			tTimeToDose := REAL_TO_TIME( (UINT_TO_REAL(nDoseQtyMls) * 1000.0) / (UINT_TO_REAL(nDoseRateMLph) / 60.0 / 60.0 ));
			fbTONdoseTime.IN := FALSE;
			fbTONdoseTime.PT := tTimeToDose;
			fbTONdoseTime.IN := TRUE;
			eState := E_DeviceState.RUNNING;
			bBusy := TRUE;
			eSMState := WAIT;
		END_IF
		
		IF fbTONdoseTime.Q THEN
			eStateTarget := E_DeviceState.IDLE;
			eState := E_DeviceState.IDLE;
			bBusy := FALSE;
		END_IF
			
	END_IF

{warning 'add method implementation '}
METHOD disable : BOOL
bEnable := False;
END_METHOD

{warning 'add method implementation '}
METHOD enable : BOOL
bEnable := True;
END_METHOD

{warning 'add method implementation '}
METHOD executeDose : BOOL
VAR_INPUT
	DoseQtyMls	: UINT;
	DoseRateMlph	: UINT;
	RequestComplete	: POINTER TO BOOL;
END_VAR
VAR_OUTPUT
	RequestAccepted	: BOOL;
END_VAR
IF bBusy = FALSE THEN
	IF bEnable THEN
		nDoseQtyMls := DoseQtyMls;
		nDoseRateMLph := DoseRateMLph;
		tTimeToDose := REAL_TO_TIME( (UINT_TO_REAL(nDoseQtyMls) * 1000.0) / (UINT_TO_REAL(DoseRateMLph) / 60.0 / 60.0 ));
		RequestAccepted := TRUE;
		bRequestSentToMaster := FALSE;
		bRequestFinished := RequestComplete;
		eSMState := SET_DOSE_TRIG;
		executeDose := TRUE;
	END_IF
ELSE
	executeDose := FALSE;
END_IF
END_METHOD

METHOD FB_init : BOOL
VAR_INPUT
	bInitRetains : BOOL; // if TRUE, the retain variables are initialized (warm start / cold start)
	bInCopyCode : BOOL;  // if TRUE, the instance afterwards gets moved into the copy code (online change)
	
	MotorID: STRING;
	MotorDescr: STRING;
	
	ModbusUnitID: UINT; 
	//ModbusMaster: FB_ModbusMaster;
	
END_VAR
sID := MotorID;
sDescr := MotorDescr;
nModbusUnitID := ModbusUnitID;
//fbModbusMaster := ModbusMaster;
END_METHOD

METHOD readReg : BOOL
VAR_INPUT
	RequestComplete	: POINTER TO BOOL;
	AddressToRead: UINT;
	NumberWords: UINT;
END_VAR
VAR_OUTPUT
	RequestAccepted	: BOOL;
END_VAR
IF bBusy = FALSE THEN
	IF bEnable THEN
		nReadRegsVals[1] := 16#00;
		nReadRegsVals[2] := 16#00;
		nReadRegsVals[3] := 16#00;
		nReadRegsVals[4] := 16#00;
		nRegisterWordstoRead := NumberWords;
		nAddrRead:= AddressToRead;
		eSMState := READ_TRIG;
		bBusy := TRUE;		
		readReg := TRUE;		
	END_IF
ELSE
	readReg := FALSE;
END_IF
END_METHOD

METHOD resetStatistics : BOOL
VAR_INPUT
END_VAR
END_METHOD

{warning 'add method implementation '}
METHOD setBatch : BOOL
VAR_INPUT
	BatchQtyMl	: UINT;
	RequestComplete	: POINTER TO BOOL;
END_VAR
VAR_OUTPUT
	RequestAccepted	: BOOL;
END_VAR

VAR
	SET_BATCH_QTY_TRIG: E_DeviceState;
END_VAR
IF bBusy = FALSE THEN
	IF bEnable THEN
		nBatchQtyMl := BatchQtyMl;
		RequestAccepted := TRUE;
		bRequestSentToMaster := FALSE;
		bRequestFinished := RequestComplete;
		eSMState := SET_BATCH_QTY_TRIG;
		setBatch := TRUE;
	END_IF
ELSE 
	setBatch := FALSE;
END_IF
END_METHOD

METHOD setCapacity : BOOL
VAR_INPUT
	Capacity: DINT;
END_VAR
VAR_INPUT
	RequestComplete	: POINTER TO BOOL;
END_VAR
VAR_OUTPUT
	RequestAccepted	: BOOL;
END_VAR
IF bBusy = FALSE THEN
	IF bEnable THEN
		nWriteRegsVals[1] := DINT_TO_WORD(Capacity);
		nQtyWordsWrite := 1;
		nAddrWrite := 16#C1;
		eSMState := WRITE_TRIG;
		bBusy := TRUE;		
		setCapacity := TRUE;		
	END_IF
ELSE
	setCapacity := FALSE;
END_IF
END_METHOD

METHOD setDoseParams : BOOL
VAR_INPUT
	DoseQtyMls	: UINT;
	DoseRateMlph	: UINT;
END_VAR

nDoseQtyMls := DoseQtyMls;
nDoseRateMLph := DoseRateMlph;
END_METHOD

METHOD setModbusMaster : BOOL
VAR_INPUT
	ModbusMaster: FB_ModbusMaster;
END_VAR

fbModbusMaster REF= ModbusMaster;
END_METHOD

{warning 'add method implementation '}
METHOD setOFF : BOOL
VAR_INPUT
	RequestComplete	: POINTER TO BOOL;
END_VAR
VAR_OUTPUT
	RequestAccepted	: BOOL;
END_VAR
IF bBusy = FALSE THEN
	IF bEnable THEN
		nWriteRegsVals[1] := 16#0;
		nQtyWordsWrite := 1;
		nAddrWrite := 16#8C;
		eSMState := WRITE_TRIG;
		bBusy := TRUE;		
		setOFF := TRUE;		
	END_IF
ELSE
	setOFF := FALSE;
END_IF
END_METHOD

{warning 'add method implementation '}
METHOD setON : BOOL
VAR_INPUT
	RateMlph	: UINT;
	RequestComplete	: POINTER TO BOOL;
END_VAR
VAR_OUTPUT
	RequestAccepted	: BOOL;
END_VAR
IF bBusy = FALSE AND bEnable THEN
	nWriteRegsVals[1] := 16#1;
	nQtyWordsWrite := 1;
	nAddrWrite := 16#8C;		// Emec have 2 different Modbus register schemes (check which version the pumps are and amend if necessary)
	eSMState := WRITE_TRIG;
	bBusy := TRUE;
	setON := TRUE;
ELSE
	setON := FALSE;
END_IF
END_METHOD

METHOD writeReg : BOOL
VAR_INPUT
	RequestComplete	: POINTER TO BOOL;
	Register: WORD;
	Value: WORD;
END_VAR
VAR_OUTPUT
	RequestAccepted	: BOOL;
END_VAR
IF bBusy = FALSE THEN
	IF bEnable THEN
		nWriteRegsVals[1] := Value;
		nQtyWordsWrite := 1;
		nAddrWrite := Register;
		eSMState := WRITE_TRIG;
		bBusy := TRUE;				
	END_IF
END_IF
END_METHOD

END_FUNCTION_BLOCK

// ---- POUs/99 Utilities/_ss/FB_ModbusMaster.TcPOU
FUNCTION_BLOCK FB_ModbusMaster

VAR
	MB: ModbusRtuMaster_KL6x22B;
	
	nReadRegsVals: POINTER TO ARRAY[1..10] OF WORD;
	nWriteRegVals: ARRAY[1..10] OF WORD;
	
	
	bRequestFinshed : POINTER TO BOOL;
		
	nSlaveAddress : BYTE;
	nQtyWordsToRead : WORD;
	nQtyWordsToWrite : WORD;
	nAdrFirstSlaveRegisterRead : WORD;
	nAdrFirstSlaveRegisterWrite : WORD;
	nTimeout : TIME := T#5S;
	
	
	// State Machine
	eState: (IDLE, BUSY, ERROR) := IDLE;
	eSMtate: (WAIT, READ_TRIG, READ, WRITE_TRIG, WRITE, ERROR) := WAIT;
	eSMState_prev:  (WAIT, READ_TRIG, READ, WRITE_TRIG, WRITE, ERROR) := WAIT;
	bBusy: BOOL;
	
	//eOperationType: (READ_OP, WRITE_OP, READWRITE_OP);
	eOperationType: E_AccessType;
	fbTrigger : R_TRIG;
	
	bOperationFirstRun: BOOL := TRUE;
	nNumRetries: INT := 0; 
	nRetryThreshold: INT := 10;

END_VAR

fbTrigger();

CASE eState OF
	WAIT :
		eState := IDLE;
		MB.ReadRegs(Execute := FALSE);
        MB.WriteRegs(Execute := FALSE);
	
		
		IF fbTrigger.Q THEN
			IF eOperationType = E_AccessType.WRITE THEN
				eSMtate := WRITE_TRIG;
			ELSIF eOperationType = E_AccessType.READ THEN
				eSMtate := READ_TRIG;
			END_IF
		END_IF
		
		
		
	READ_TRIG : 
		eState := BUSY;
		IF bOperationFirstRun THEN
			nNumRetries := 0;
			bOperationFirstRun := FALSE;
		END_IF
	
		IF eOperationType = E_AccessType.READ THEN
			
			 MB.ReadRegs(
				UnitID:= nSlaveAddress, 
				Quantity:= nQtyWordsToRead, 
				MBAddr:= nAdrFirstSlaveRegisterRead, 
				cbLength:= nQtyWordsToRead * 2,//SIZEOF(nReadRegsVals), 
				pMemoryAddr:= ADR(nReadRegsVals), 
				Execute:= TRUE, 
				Timeout:= nTimeout );
			
			
			IF NOT MB.BUSY THEN 
				MB.ReadRegs(Execute := FALSE );
				bBusy := TRUE;
				IF MB.Error THEN 
					eSMState_prev := eSMtate;
					eSMtate := ERROR;           // handle errors 
				ELSE 
					eSMtate := READ; // [...]               // keep going 
				END_IF
			END_IF
		END_IF
		
		
	READ :
	
		IF NOT MB.BUSY THEN
			eSMtate := WAIT;
			bRequestFinshed^ := TRUE;
			bBusy := FALSE;
			fbTrigger.CLK := FALSE;
			bOperationFirstRun := TRUE;
		ELSIF MB.Error THEN
			eSMState_prev := eSMtate;
			eSMtate := ERROR;
		END_IF
	
	
	
	WRITE_TRIG :

		IF bOperationFirstRun THEN
			nNumRetries := 0;
			bOperationFirstRun := FALSE;
		END_IF
	(*
		MB.WriteRegs(
			UnitID:= nSlaveAddress, 
			Quantity:= nQtyWordsToWrite, 
			MBAddr:= nAdrFirstSlaveRegisterWrite, 
			cbLength:= nQtyWordsToWrite * 2, 
			pMemoryAddr:= ADR(nWriteRegVals), 
			Execute:= TRUE, 
			Timeout:= nTimeout); 
		*)	
		
		MB.UnitID:= nSlaveAddress;
		MB.Quantity:=1;
		MB.MBAddr:= nAdrFirstSlaveRegisterWrite;
		MB.cbLength:= nQtyWordsToWrite * 2;
		MB.pMemoryAddr:= ADR(nWriteRegVals);
		MB.Execute:= TRUE;
		MB.Timeout:= nTimeout;
		MB.WriteSingleRegister();
		
			
		IF NOT MB.BUSY THEN 
			//MB.WriteRegs(Execute := FALSE );
			MB.Execute := FALSE;
			bBusy := TRUE;
			IF MB.Error THEN 
				eSMState_prev := eSMtate;
				eSMtate := ERROR;           				// handle errors 
			ELSE 
				eSMtate := WRITE;			            // keep going 
			END_IF
		END_IF

	
		
	WRITE:
		IF NOT MB.BUSY THEN
			eSMtate := WAIT;
			bRequestFinshed^ := TRUE;
			bBusy := FALSE;
			fbTrigger.CLK := FALSE;
			bOperationFirstRun := TRUE;
		ELSIF MB.Error THEN
			eSMState_prev := eSMtate;
			eSMtate := ERROR;
		END_IF
	
		
	ERROR:
		nNumRetries := nNumRetries + 1;
		IF nNumRetries > nRetryThreshold THEN
			eState := ERROR;
		ELSE
			eSMtate := eSMState_prev;
		END_IF
		 
			
		

END_CASE

METHOD Error : BOOL
VAR_INPUT
END_VAR
Error := MB.Error;
END_METHOD

METHOD FB_init : BOOL
VAR_INPUT
	bInitRetains : BOOL; // if TRUE, the retain variables are initialized (warm start / cold start)
	bInCopyCode : BOOL;  // if TRUE, the instance afterwards gets moved into the copy code (online change)
END_VAR
END_METHOD

METHOD isBusy : BOOL
isBusy := bBusy;
END_METHOD

METHOD readRegs : BOOL
VAR_INPUT
	
	ReadRegsVals: POINTER TO ARRAY[1..10] OF WORD;
	SlaveAddress : UINT;
	QtyWordsToRead : UINT;
	AdrFirstSlaveRegisterRead : UINT;
	bRequestCompleted : POINTER TO BOOL;
	
END_VAR

VAR_OUTPUT
	bRequestAccepted: BOOL;
END_VAR
IF eState = WAIT THEN
	eOperationType := E_AccessType.READ;
	nReadRegsVals := ReadRegsVals;
	nSlaveAddress := UINT_TO_BYTE(SlaveAddress);
	nQtyWordsToRead := UINT_TO_WORD(QtyWordsToRead);
	nAdrFirstSlaveRegisterRead := UINT_TO_WORD(AdrFirstSlaveRegisterRead);
	fbTrigger.CLK := TRUE;
	bRequestAccepted := TRUE;
	bBusy := TRUE;
	bRequestFinshed := bRequestCompleted;
END_IF
END_METHOD

METHOD writeReg : BOOL
VAR_INPUT
	WriteRegVal: WORD;
	SlaveAddress : UINT;
	AdrFirstSlaveRegisterWrite : UINT;
	bRequestCompleted : POINTER TO BOOL;
END_VAR

VAR_OUTPUT
	bRequestAccepted: BOOL := FALSE;
END_VAR

IF eState = WAIT THEN
	eOperationType := E_AccessType.WRITE;
	nWriteRegVals[1] := WriteRegVal;
	nSlaveAddress := UINT_TO_BYTE(SlaveAddress);
	nQtyWordsToWrite := 1;
	nAdrFirstSlaveRegisterWrite := UINT_TO_BYTE(AdrFirstSlaveRegisterWrite);
	bRequestAccepted := TRUE;
	bRequestFinshed := bRequestCompleted;
	fbTrigger.CLK := TRUE;
	eState := WRITE_TRIG;
	
END_IF
END_METHOD

METHOD writeRegs : BOOL
VAR_INPUT

	WriteRegVals: ARRAY[1..10] OF WORD;
	
	SlaveAddress : UINT;
	QtyWordsToWrite : UINT;
	AdrFirstSlaveRegisterWrite : UINT;
	bRequestCompleted: POINTER TO BOOL;

END_VAR

VAR_OUTPUT
	bRequestAccepted: BOOL := FALSE;
END_VAR
IF eState = WAIT THEN
	eOperationType := E_AccessType.WRITE;
	nWriteRegVals := WriteRegVals;
	nSlaveAddress := UINT_TO_BYTE(SlaveAddress);
	nQtyWordsToWrite := UINT_TO_WORD(QtyWordsToWrite);
	nAdrFirstSlaveRegisterWrite := UINT_TO_WORD(AdrFirstSlaveRegisterWrite);
	fbTrigger.CLK := TRUE;
	bRequestAccepted := TRUE;
	bRequestFinshed := bRequestCompleted;
	eState := WRITE_TRIG;
END_IF
END_METHOD

END_FUNCTION_BLOCK

// ---- POUs/01 Actuators/Dosing Machine/FB_DrumFilter_Faivre120.TcPOU
{attribute 'OPC.UA.DA.StructuredType' := '1'}
FUNCTION_BLOCK FB_DrumFilter_Faivre120 EXTENDS FB_BaseDevice IMPLEMENTS I_Device

VAR
	
	{attribute 'OPC.UA.DA' := '1'}   
	bInContactor AT %I*: BOOL := FALSE;
	{attribute 'OPC.UA.DA' := '1'}   
	bOutContactor AT %Q*: BOOL := FALSE;
	{attribute 'OPC.UA.DA' := '1'}   
	bInMCCB AT %I*: BOOL := FALSE;
	{attribute 'OPC.UA.DA' := '1'}   
	bInRunning AT %I*: BOOL := FALSE;
	{attribute 'OPC.UA.DA' := '1'}   
	bInFault_Motors AT %I*: BOOL := FALSE;
	{attribute 'OPC.UA.DA' := '1'}   
	bInFault_Overflow AT %I*: BOOL := FALSE;
	{attribute 'OPC.UA.DA' := '0'}   
	eSMState: (WAIT, TURNING_ON, ON, TURNING_OFF, OFF);
	{attribute 'OPC.UA.DA' := '0'}   
	tActionTimeout: TIME := T#5S;
	{attribute 'OPC.UA.DA' := '0'}   
	fbTON_timeout: TON := (PT := tActionTimeout, IN := FALSE);
	{attribute 'OPC.UA.DA' := '0'}  
	fbTON_simulation_delay: TON := (PT := T#1S, IN := FALSE);
END_VAR

fbTONstartTime();
fbTONstopTime();


IF GVL.bAutoUpdateDeviceState THEN
	eState := eStateTarget;	
END_IF


IF eMode <> E_DeviceMode.SIMULATION THEN
	
	
	IF bEnable THEN
		IF eStateTarget = E_DeviceState.ON AND eState <> E_DeviceState.ON THEN
			eSMState := TURNING_ON;
		END_IF
	END_IF
	
	IF eStateTarget = E_DeviceState.OFF AND eState <> E_DeviceState.OFF THEN
			eSMState := TURNING_OFF;
	END_IF
	
	
	CASE eSMState OF
		
		WAIT:
			//Wait for method call to change ESMState
			
		TURNING_ON: 
			eState := E_DeviceState.TURNING_ON;
	
			bOutContactor := TRUE;
		
			IF fbTONstartTime.Q THEN
				eSMState := WAIT;
				raiseAlarm(Priority := E_AlarmPriority.High, Label := 'Failed to Start', Enabled := TRUE, DeviceAlarmID := 1);
			END_IF
			
			IF bInContactor  THEN
				eSMState := ON;
				eState := E_DeviceState.ON;
			END_IF
			
		ON:
			IF bInContactor <> TRUE THEN
				raiseAlarm(Priority := E_AlarmPriority.High, Label := 'Power Lost', Enabled := TRUE, DeviceAlarmID := 2);
				eState := E_DeviceState.OFF;
				eSMState := WAIT;
			END_IF
			
	
			
		TURNING_OFF:
			eState := E_DeviceState.TURNING_OFF;
			bOutContactor := FALSE;
	
					
			IF fbTONstopTime.Q THEN
				eSMState := WAIT;
				raiseAlarm(Priority := E_AlarmPriority.High, Label := 'Failed to Stop', Enabled := TRUE,  DeviceAlarmID := 3);
			END_IF 
			
			IF bInContactor = FALSE THEN
				eSMState := OFF;	
			END_IF
	
			
			
		OFF:
			eState := E_DeviceState.OFF;
			eSMState := WAIT;
			
			
	END_CASE
	
	
(*
				SIMULATION CODE 
				This code forces the contactor feedback ON or OFF depending on whether the device has been told to turn on or off
*)

ELSIF eMode = E_DeviceMode.SIMULATION THEN
	
fbTON_simulation_delay();
	
	IF eSMState = TURNING_ON THEN  					
		fbTON_simulation_delay.IN := TRUE;
		IF fbTON_simulation_delay.Q THEN
			bInContactor := TRUE;
			fbTON_simulation_delay.IN := FALSE;	
		END_IF
		
	ELSIF eSMState = TURNING_OFF THEN
		fbTON_simulation_delay.IN := TRUE;
		IF fbTON_simulation_delay.Q THEN
			bInContactor := FALSE;
			fbTON_simulation_delay.IN := FALSE;	
		END_IF
	END_IF
END_IF

{warning 'add method implementation '}
METHOD disable : BOOL
bEnable := FALSE;
END_METHOD

{warning 'add method implementation '}
METHOD enable : BOOL
bEnable := TRUE;
END_METHOD

METHOD FB_init : BOOL
VAR_INPUT
	bInitRetains : BOOL; // if TRUE, the retain variables are initialized (warm start / cold start)
	bInCopyCode : BOOL;  // if TRUE, the instance afterwards gets moved into the copy code (online change)
	
	FilterID: STRING(80);
	FIlterDescr: STRING(255);
END_VAR
sID := FilterID;
sDescr := FIlterDescr;
END_METHOD

METHOD setOff : BOOL
VAR_INPUT
END_VAR
eSMState := TURNING_OFF;
fbTONstopTime.IN := TRUE;
bBusy := FALSE;
END_METHOD

METHOD setOn : BOOL
VAR_INPUT
END_VAR
eSMState := TURNING_ON;
fbTONstartTime.IN := TRUE;
bBusy := TRUE;
END_METHOD

END_FUNCTION_BLOCK

// ---- POUs/01 Actuators/Dosing Machine/FB_DrumFilter_Faivre60.TcPOU
{attribute 'OPC.UA.DA.StructuredType' := '1'}
FUNCTION_BLOCK FB_DrumFilter_Faivre60 EXTENDS FB_BaseDevice IMPLEMENTS I_Device

VAR

	{attribute 'OPC.UA.DA' := '1'}   
	bInContactor AT %I*: BOOL := FALSE;
	{attribute 'OPC.UA.DA' := '1'}   
	bOutContactor AT %Q*: BOOL := FALSE;
	{attribute 'OPC.UA.DA' := '1'}   
	bInMCCB AT %I*: BOOL := FALSE;
	{attribute 'OPC.UA.DA' := '1'}   
	bInRunning AT %I*: BOOL := FALSE;
	{attribute 'OPC.UA.DA' := '1'}   
	bInFault_Motors AT %I*: BOOL := FALSE;
	{attribute 'OPC.UA.DA' := '1'}   
	bInFault_Overflow AT %I*: BOOL := FALSE;
	{attribute 'OPC.UA.DA' := '0'}   
	eSMState: (WAIT, TURNING_ON, ON, TURNING_OFF, OFF);
	{attribute 'OPC.UA.DA' := '0'}   
	tActionTimeout: TIME := T#5S;
	{attribute 'OPC.UA.DA' := '0'}   
	fbTON_timeout: TON := (PT := tActionTimeout, IN := FALSE);
	{attribute 'OPC.UA.DA' := '0'}
	fbTON_simulation_delay: TON := (PT := T#1S, IN := FALSE);
END_VAR

fbTONstartTime();
fbTONstopTime();

IF GVL.bAutoUpdateDeviceState THEN
	eState := eStateTarget;	
END_IF

IF eMode <> E_DeviceMode.SIMULATION THEN
	
	
	
	
	IF bEnable THEN
		IF eStateTarget = E_DeviceState.ON AND eState <> E_DeviceState.ON THEN
			eSMState := TURNING_ON;
		END_IF
	END_IF
	
	IF eStateTarget = E_DeviceState.OFF AND eState <> E_DeviceState.OFF THEN
			eSMState := TURNING_OFF;
	END_IF
	
	
	CASE eSMState OF
		
		WAIT:
			//Wait for method call to change ESMState
			
		TURNING_ON: 
			eState := E_DeviceState.TURNING_ON;
	
			bOutContactor := TRUE;
		
			IF fbTONstartTime.Q THEN
				eSMState := WAIT;
				raiseAlarm(Priority := E_AlarmPriority.High, Label := 'Failed to Start', Enabled := TRUE, DeviceAlarmID := 1);
			END_IF
			
			IF bInContactor  THEN
				eSMState := ON;
				eState := E_DeviceState.ON;
			END_IF
			
		ON:
			IF bInContactor <> TRUE THEN
				raiseAlarm(Priority := E_AlarmPriority.High, Label := 'Power Lost', Enabled := TRUE, DeviceAlarmID := 2);
				eState := E_DeviceState.OFF;
				eSMState := WAIT;
			END_IF
			
	
			
		TURNING_OFF:
			eState := E_DeviceState.TURNING_OFF;
			bOutContactor := FALSE;
	
					
			IF fbTONstopTime.Q THEN
				eSMState := WAIT;
				raiseAlarm(Priority := E_AlarmPriority.High, Label := 'Failed to Stop', Enabled := TRUE, DeviceAlarmID := 3);
			END_IF 
			
			IF bInContactor = FALSE THEN
				eSMState := OFF;	
			END_IF
			
	
		OFF:
			eState := E_DeviceState.OFF;
			eSMState := WAIT;
			
			
	END_CASE
	
(*
				SIMULATION CODE 
				This code forces the contactor feedback ON or OFF depending on whether the device has been told to turn on or off
*)

ELSIF eMode = E_DeviceMode.SIMULATION THEN
	
fbTON_simulation_delay();
	
	IF eSMState = TURNING_ON THEN  					
		fbTON_simulation_delay.IN := TRUE;
		IF fbTON_simulation_delay.Q THEN
			bInContactor := TRUE;
			fbTON_simulation_delay.IN := FALSE;	
		END_IF
		
	ELSIF eSMState = TURNING_OFF THEN
		fbTON_simulation_delay.IN := TRUE;
		IF fbTON_simulation_delay.Q THEN
			bInContactor := FALSE;
			fbTON_simulation_delay.IN := FALSE;	
		END_IF
	END_IF
END_IF

{warning 'add method implementation '}
METHOD disable : BOOL
bEnable := FALSE;
END_METHOD

{warning 'add method implementation '}
METHOD enable : BOOL
bEnable := TRUE;
END_METHOD

METHOD FB_init : BOOL
VAR_INPUT
	bInitRetains : BOOL; // if TRUE, the retain variables are initialized (warm start / cold start)
	bInCopyCode : BOOL;  // if TRUE, the instance afterwards gets moved into the copy code (online change)
	
	FilterID: STRING(80);
	FIlterDescr: STRING(255);
END_VAR
sID := FilterID;
sDescr := FIlterDescr;
END_METHOD

METHOD setOff : BOOL
VAR_INPUT
END_VAR
eSMState := TURNING_OFF;
bBusy := FALSE;
END_METHOD

METHOD setOn : BOOL
VAR_INPUT
END_VAR
eSMState := TURNING_ON;
bBusy := TRUE;
END_METHOD

END_FUNCTION_BLOCK

// ---- POUs/01 Actuators/Dosing Machine/FB_GasMonitoringPanel_CDA4022.TcPOU
{attribute 'OPC.UA.DA.StructuredType' := '1'}
FUNCTION_BLOCK FB_GasMonitoringPanel_CDA4022 EXTENDS FB_BaseDevice 

VAR_IN_OUT
	{attribute 'OPC.UA.DA' := '0'}
	fbModbusMaster: FB_ModbusMaster;
END_VAR

VAR
	// CDA Panel 4022 V3.0 Variables (https://drive.google.com/file/d/1dn1Ot7nd1VML-1RxFooYWTdx5gniYgca/view?usp=sharing)
	(*
	       CO2
		   References - https://iceblast.com.au/wp-content/uploads/2021/03/ABCB-Handbook-Indoor-Air-Quality-2018.pdf   
	*)
	nConcentration_CO2: 	UINT; // reading is value x 10, units are configurable - set to ppm
	nThreshold_CO2_Level1: 	DINT := 800; //ppm (Upper limit of AS 1668.2 recommendation (for CO2 controlled ventilation))
	nAlarm_CO2_Level1: 		UINT; 
	nThreshold_CO2_Level2: 	DINT := 1000; //ppm (ASHRAE 62.1 recommendation (occupant comfort))
	nAlarm_CO2_Level2: 		UINT; 
	nThreshold_CO2_Level3: 	DINT := 5000; //ppm (Australian occupational exposure limit (SWA 2011b) )
	nAlarm_CO2_Level3: 		UINT; 
	
	(*
	       O2
		   References - https://www.cacgas.com.au/blog/bid/378107/oxygen-o2-occupational-health-exposure-standards 
	*)
	nConcentration_O2: 		UINT; // reading is value x 10, units are configurable - set to ppm
	nThreshold_O2_Level1: 	DINT := 195000; //ppm (Minimum "Safe Level")
	nAlarm_O2_Level1: 		UINT; 
	nThreshold_O2_Level2: 	DINT := 160000; //ppm (First signs of anoxia (dizziness, light-headedness))
	nAlarm_O2_Level2: 		UINT; 
	nThreshold_O2_Level3: 	DINT := 235000; //ppm (oxygen levels that exceed 23.5% present a serious fire danger.  At levels of 25%+ items such as clothing can spontaneously combust.  )
	nAlarm_O2_Level3: 		UINT; 	


	// Modbus Variables
	nModbusUnitID: UINT; 
	
	nPointerInt: POINTER TO INT;  // used to 
	
	{attribute 'OPC.UA.DA' := '0'}
	nReadRegsVals: ARRAY[1..10] OF WORD;
	{attribute 'OPC.UA.DA' := '0'}
	nWriteRegsVals: ARRAY[1..10] OF WORD;
	{attribute 'OPC.UA.DA' := '0'}
	nQtyWordsWrite: UINT;
	{attribute 'OPC.UA.DA' := '0'}
	nAddrWrite: UINT;
	{attribute 'OPC.UA.DA' := '0'}
	nRegisterWordstoRead: UINT;
	{attribute 'OPC.UA.DA' := '0'}
	nAddrRead: UINT;
	
	// Async Statemachine Variables
	{attribute 'OPC.UA.DA' := '0'}
	eSMState: (WAIT, READ_TRIG, READ, WRITE_TRIG, WRITE, ERROR);
	{attribute 'OPC.UA.DA' := '0'} 
	eOpType: (READ_OP, WRITE_OP);
	{attribute 'OPC.UA.DA' := '0'} 
	bRequestFinished: POINTER TO BOOL;
	{attribute 'OPC.UA.DA' := '0'} 
	bRequestSentToMaster: BOOL 	:= FALSE;
	{attribute 'OPC.UA.DA' := '0'} 
	bRequestCompleted: BOOL 	:= FALSE;
	


	
END_VAR


IF GVL.bAutoUpdateDeviceState THEN
	eState := eStateTarget;	
END_IF


CASE eSMState OF
	
	WAIT :
	//Do nothing and wait for eState to be changed by a called method

	READ_TRIG : 
	
		fbModbusMaster.readRegs(
			ReadRegsVals:= ADR(nPointerInt^), 
			SlaveAddress:= nModbusUnitID, 
			QtyWordsToRead:= nRegisterWordstoRead, 
			AdrFirstSlaveRegisterRead:= nAddrRead, 
			bRequestCompleted:= ADR(bRequestCompleted), 
			bRequestAccepted=> bRequestSentToMaster);
				
		IF bRequestSentToMaster THEN
			eSMState := READ;				
		END_IF
	
	READ:
		IF bRequestCompleted THEN	
			eSMState := WAIT; 			
			bRequestSentToMaster := FALSE;
			bRequestCompleted := FALSE;
			bBusy := FALSE;
		END_IF
		

	WRITE_TRIG :
		
		fbModbusMaster.writeReg(
			WriteRegVal := nWriteRegsVals[1],
			SlaveAddress := nModbusUnitID,
			AdrFirstSlaveRegisterWrite := nAddrWrite,
			bRequestCompleted := ADR(bRequestCompleted),
			bRequestAccepted => bRequestSentToMaster);
			
		IF bRequestSentToMaster THEN
			eSMState := WRITE;           
		END_IF
		
	WRITE:
		IF bRequestCompleted THEN
			eSMState := WAIT;
			bRequestCompleted := FALSE;
			bRequestSentToMaster := FALSE;
			bBusy := FALSE;
		END_IF
END_CASE

METHOD FB_init : BOOL
VAR_INPUT
	bInitRetains : BOOL; // if TRUE, the retain variables are initialized (warm start / cold start)
	bInCopyCode : BOOL;  // if TRUE, the instance afterwards gets moved into the copy code (online change)
	
	ModbusID: UINT;
END_VAR
nModbusUnitID := ModbusID;
END_METHOD

METHOD read_Alarm_CO2_Lvl1 : BOOL
VAR_INPUT
END_VAR
IF NOT bBusy AND bEnable THEN
	nPointerInt := ADR(nAlarm_CO2_Level1);
	nRegisterWordstoRead := 1;
	nAddrRead:= 101;
	eSMState := READ_TRIG;
	bBusy := TRUE;		
	read_Alarm_CO2_Lvl1 := TRUE;		
ELSE
	read_Alarm_CO2_Lvl1 := FALSE;
END_IF
END_METHOD

METHOD read_Alarm_CO2_Lvl2 : BOOL
VAR_INPUT
END_VAR
IF NOT bBusy AND bEnable THEN
	nPointerInt := ADR(nAlarm_CO2_Level2);
	nRegisterWordstoRead := 1;
	nAddrRead:= 201;
	eSMState := READ_TRIG;
	bBusy := TRUE;		
	read_Alarm_CO2_Lvl2 := TRUE;		
ELSE
	read_Alarm_CO2_Lvl2 := FALSE;
END_IF
END_METHOD

METHOD read_Alarm_CO2_Lvl3 : BOOL
VAR_INPUT
END_VAR
IF NOT bBusy AND bEnable THEN
	nPointerInt := ADR(nAlarm_CO2_Level3);
	nRegisterWordstoRead := 1;
	nAddrRead:= 301;
	eSMState := READ_TRIG;
	bBusy := TRUE;		
	read_Alarm_CO2_Lvl3 := TRUE;		
ELSE
	read_Alarm_CO2_Lvl3 := FALSE;
END_IF
END_METHOD

METHOD read_Alarm_O2_Lvl1 : BOOL
VAR_INPUT
END_VAR
IF NOT bBusy AND bEnable THEN
	nPointerInt := ADR(nAlarm_O2_Level1);
	nRegisterWordstoRead := 1;
	nAddrRead:= 100;
	eSMState := READ_TRIG;
	bBusy := TRUE;		
	read_Alarm_O2_Lvl1 := TRUE;		
ELSE
	read_Alarm_O2_Lvl1 := FALSE;
END_IF
END_METHOD

METHOD read_Alarm_O2_Lvl2 : BOOL
VAR_INPUT
END_VAR
IF NOT bBusy AND bEnable THEN
	nPointerInt := ADR(nAlarm_O2_Level2);
	nRegisterWordstoRead := 1;
	nAddrRead:= 200;
	eSMState := READ_TRIG;
	bBusy := TRUE;		
	read_Alarm_O2_Lvl2 := TRUE;		
ELSE
	read_Alarm_O2_Lvl2 := FALSE;
END_IF
END_METHOD

METHOD read_Alarm_O2_Lvl3 : BOOL
VAR_INPUT
END_VAR
IF NOT bBusy AND bEnable THEN
	nPointerInt := ADR(nAlarm_O2_Level3);
	nRegisterWordstoRead := 1;
	nAddrRead:= 300;
	eSMState := READ_TRIG;
	bBusy := TRUE;		
	read_Alarm_O2_Lvl3 := TRUE;		
ELSE
	read_Alarm_O2_Lvl3 := FALSE;
END_IF
END_METHOD

METHOD read_Concentration_CO2 : BOOL
VAR_INPUT
END_VAR
IF NOT bBusy AND bEnable THEN
	nPointerInt := ADR(nConcentration_CO2);
	nRegisterWordstoRead := 1;
	nAddrRead:= 1;
	eSMState := READ_TRIG;
	bBusy := TRUE;		
	read_Concentration_CO2 := TRUE;		
ELSE
	read_Concentration_CO2 := FALSE;
END_IF
END_METHOD

METHOD read_Concentration_O2 : BOOL
VAR_INPUT
END_VAR
IF NOT bBusy AND bEnable THEN
	nPointerInt := ADR(nConcentration_O2);
	nRegisterWordstoRead := 1;
	nAddrRead:= 0;
	eSMState := READ_TRIG;
	bBusy := TRUE;		
	read_Concentration_O2 := TRUE;		
ELSE
	read_Concentration_O2 := FALSE;
END_IF
END_METHOD

END_FUNCTION_BLOCK

// ---- POUs/01 Actuators/Dosing Machine/FB_GasMonitoringPanel_CDA4022_R2.TcPOU
{attribute 'OPC.UA.DA.StructuredType' := '1'}
FUNCTION_BLOCK FB_GasMonitoringPanel_CDA4022_R2 EXTENDS FB_BaseDevice 

VAR_IN_OUT
	{attribute 'OPC.UA.DA' := '0'}
	fbModbusManager: FB_ModbusManager;
END_VAR

VAR
	// CDA Panel 4022 V3.0 Variables (https://drive.google.com/file/d/1dn1Ot7nd1VML-1RxFooYWTdx5gniYgca/view?usp=sharing)
	(*
	       CO2
		   References - https://iceblast.com.au/wp-content/uploads/2021/03/ABCB-Handbook-Indoor-Air-Quality-2018.pdf   
	*)
	nConcentration_CO2: 	UINT; // reading is value x 10, units are configurable - set to ppm
	nThreshold_CO2_Level1: 	DINT := 800; //ppm (Upper limit of AS 1668.2 recommendation (for CO2 controlled ventilation))
	nAlarm_CO2_Level1: 		UINT; 
	nThreshold_CO2_Level2: 	DINT := 1000; //ppm (ASHRAE 62.1 recommendation (occupant comfort))
	nAlarm_CO2_Level2: 		UINT; 
	nThreshold_CO2_Level3: 	DINT := 5000; //ppm (Australian occupational exposure limit (SWA 2011b) )
	nAlarm_CO2_Level3: 		UINT; 
	
	(*
	       O2
		   References - https://www.cacgas.com.au/blog/bid/378107/oxygen-o2-occupational-health-exposure-standards 
	*)
	nConcentration_O2: 		UINT; // reading is value x 10, units are configurable - set to ppm
	nThreshold_O2_Level1: 	DINT := 195000; //ppm (Minimum "Safe Level")
	nAlarm_O2_Level1: 		UINT; 
	nThreshold_O2_Level2: 	DINT := 160000; //ppm (First signs of anoxia (dizziness, light-headedness))
	nAlarm_O2_Level2: 		UINT; 
	nThreshold_O2_Level3: 	DINT := 235000; //ppm (oxygen levels that exceed 23.5% present a serious fire danger.  At levels of 25%+ items such as clothing can spontaneously combust.  )
	nAlarm_O2_Level3: 		UINT; 	

	// Modbus Variables
	nModbusUnitID: UINT; 
	bFirtRun: BOOL := TRUE;
	bResetTimer: BOOL := TRUE;
	
	// Async Statemachine Variables
	{attribute 'OPC.UA.DA' := '0'}
	eSMState: (WAIT, READ_TRIG, READ, WRITE_TRIG, WRITE, ERROR);
	{attribute 'OPC.UA.DA' := '0'} 
	
	fbTON_DataRefresh: TON := (PT := T#15S, IN := FALSE);
	
	stModRequest_Read_CO2_Actual: ST_Modbus_ReadRequest;
	stModRequest_Read_CO2_AL1: ST_Modbus_ReadRequest;
	stModRequest_Read_CO2_AL2: ST_Modbus_ReadRequest;
	stModRequest_Read_CO2_AL3: ST_Modbus_ReadRequest;
	
	stModRequest_Read_O2_Actual: ST_Modbus_ReadRequest;
	stModRequest_Read_O2_AL1: ST_Modbus_ReadRequest;
	stModRequest_Read_O2_AL2: ST_Modbus_ReadRequest;
	stModRequest_Read_O2_AL3: ST_Modbus_ReadRequest;
	
	
	eOpType: (READ_OP, WRITE_OP);
	{attribute 'OPC.UA.DA' := '0'} 
	bRequestFinished: POINTER TO BOOL;
	{attribute 'OPC.UA.DA' := '0'} 
	bRequestSentToMaster: BOOL 	:= FALSE;
	{attribute 'OPC.UA.DA' := '0'} 
	bRequestCompleted: BOOL 	:= FALSE;
	

	
END_VAR

fbTON_DataRefresh();

IF GVL.bAutoUpdateDeviceState THEN
	eState := eStateTarget;	
END_IF

IF bFirtRun THEN
	init_ModbusRequests();
	bFirtRun := FALSE;
END_IF

IF bResetTimer THEN
	fbTON_DataRefresh.IN := TRUE;
	bResetTimer := FALSE;
END_IF


IF fbTON_DataRefresh.Q THEN
	fbModbusManager.addRequest_Read(ReadRequest := ADR(stModRequest_Read_CO2_Actual));
	fbModbusManager.addRequest_Read(ReadRequest := ADR(stModRequest_Read_CO2_AL1));
	fbModbusManager.addRequest_Read(ReadRequest := ADR(stModRequest_Read_CO2_AL2));
	fbModbusManager.addRequest_Read(ReadRequest := ADR(stModRequest_Read_CO2_AL3));
	fbModbusManager.addRequest_Read(ReadRequest := ADR(stModRequest_Read_O2_Actual));
	fbModbusManager.addRequest_Read(ReadRequest := ADR(stModRequest_Read_O2_AL1));
	fbModbusManager.addRequest_Read(ReadRequest := ADR(stModRequest_Read_O2_AL2));
	fbModbusManager.addRequest_Read(ReadRequest := ADR(stModRequest_Read_O2_AL3));
	
	fbTON_DataRefresh.IN := FALSE;
	bResetTimer := TRUE;
END_IF

nConcentration_CO2 := WORD_TO_UINT(stModRequest_Read_CO2_Actual.ReadRegsVals[1]);
nAlarm_CO2_Level1 := WORD_TO_UINT(stModRequest_Read_CO2_AL1.ReadRegsVals[1]);
nAlarm_CO2_Level2 := WORD_TO_UINT(stModRequest_Read_CO2_AL2.ReadRegsVals[1]);
nAlarm_CO2_Level3 := WORD_TO_UINT(stModRequest_Read_CO2_AL3.ReadRegsVals[1]);

nConcentration_O2 := WORD_TO_UINT(stModRequest_Read_O2_Actual.ReadRegsVals[1]);
nAlarm_O2_Level1 := WORD_TO_UINT(stModRequest_Read_O2_AL1.ReadRegsVals[1]);
nAlarm_O2_Level2 := WORD_TO_UINT(stModRequest_Read_O2_AL2.ReadRegsVals[1]);
nAlarm_O2_Level3 := WORD_TO_UINT(stModRequest_Read_O2_AL3.ReadRegsVals[1]);

METHOD FB_init : BOOL
VAR_INPUT
	bInitRetains : BOOL; // if TRUE, the retain variables are initialized (warm start / cold start)
	bInCopyCode : BOOL;  // if TRUE, the instance afterwards gets moved into the copy code (online change)
	
	ModbusID: UINT;
END_VAR
nModbusUnitID := ModbusID;
END_METHOD

METHOD init_ModbusRequests : BOOL
VAR_INPUT
END_VAR
stModRequest_Read_CO2_Actual.SlaveAddress := nModbusUnitID;			
stModRequest_Read_CO2_Actual.AdrFirstSlaveRegisterRead := 1;
stModRequest_Read_CO2_Actual.QtyWordsToRead := 1;				// The value is a 16-bit word
stModRequest_Read_CO2_Actual.bRequestAccepted := FALSE;
stModRequest_Read_CO2_Actual.bRequestCompleted := FALSE;
stModRequest_Read_CO2_Actual.ReadRegsVals := GVL.ModbusEmptyBuffer;

stModRequest_Read_CO2_AL1.SlaveAddress := nModbusUnitID;			
stModRequest_Read_CO2_AL1.AdrFirstSlaveRegisterRead := 101;
stModRequest_Read_CO2_AL1.QtyWordsToRead := 1;				// The value is a 32-bit word
stModRequest_Read_CO2_AL1.bRequestAccepted := FALSE;
stModRequest_Read_CO2_AL1.bRequestCompleted := FALSE;
stModRequest_Read_CO2_AL1.ReadRegsVals := GVL.ModbusEmptyBuffer;

stModRequest_Read_CO2_AL2.SlaveAddress := nModbusUnitID;			
stModRequest_Read_CO2_AL2.AdrFirstSlaveRegisterRead := 201;
stModRequest_Read_CO2_AL2.QtyWordsToRead := 1;				// The value is a 32-bit word
stModRequest_Read_CO2_AL2.bRequestAccepted := FALSE;
stModRequest_Read_CO2_AL2.bRequestCompleted := FALSE;
stModRequest_Read_CO2_AL2.ReadRegsVals := GVL.ModbusEmptyBuffer;

stModRequest_Read_CO2_AL3.SlaveAddress := nModbusUnitID;			
stModRequest_Read_CO2_AL3.AdrFirstSlaveRegisterRead := 301;
stModRequest_Read_CO2_AL3.QtyWordsToRead := 1;				// The value is a 32-bit word
stModRequest_Read_CO2_AL3.bRequestAccepted := FALSE;
stModRequest_Read_CO2_AL3.bRequestCompleted := FALSE;
stModRequest_Read_CO2_AL3.ReadRegsVals := GVL.ModbusEmptyBuffer;

stModRequest_Read_O2_Actual.SlaveAddress := nModbusUnitID;			
stModRequest_Read_O2_Actual.AdrFirstSlaveRegisterRead := 0;
stModRequest_Read_O2_Actual.QtyWordsToRead := 1;				// The value is a 16-bit word
stModRequest_Read_O2_Actual.bRequestAccepted := FALSE;
stModRequest_Read_O2_Actual.bRequestCompleted := FALSE;
stModRequest_Read_O2_Actual.ReadRegsVals := GVL.ModbusEmptyBuffer;

stModRequest_Read_O2_AL1.SlaveAddress := nModbusUnitID;			
stModRequest_Read_O2_AL1.AdrFirstSlaveRegisterRead := 100;
stModRequest_Read_O2_AL1.QtyWordsToRead := 1;				// The value is a 32-bit word
stModRequest_Read_O2_AL1.bRequestAccepted := FALSE;
stModRequest_Read_O2_AL1.bRequestCompleted := FALSE;
stModRequest_Read_O2_AL1.ReadRegsVals := GVL.ModbusEmptyBuffer;

stModRequest_Read_O2_AL1.SlaveAddress := nModbusUnitID;			
stModRequest_Read_O2_AL1.AdrFirstSlaveRegisterRead := 200;
stModRequest_Read_O2_AL1.QtyWordsToRead := 1;				// The value is a 32-bit word
stModRequest_Read_O2_AL1.bRequestAccepted := FALSE;
stModRequest_Read_O2_AL1.bRequestCompleted := FALSE;
stModRequest_Read_O2_AL1.ReadRegsVals := GVL.ModbusEmptyBuffer;

stModRequest_Read_O2_AL3.SlaveAddress := nModbusUnitID;			
stModRequest_Read_O2_AL3.AdrFirstSlaveRegisterRead := 300;
stModRequest_Read_O2_AL3.QtyWordsToRead := 1;				// The value is a 32-bit word
stModRequest_Read_O2_AL3.bRequestAccepted := FALSE;
stModRequest_Read_O2_AL3.bRequestCompleted := FALSE;
stModRequest_Read_O2_AL3.ReadRegsVals := GVL.ModbusEmptyBuffer;
END_METHOD

END_FUNCTION_BLOCK

// ---- POUs/01 Actuators/Dosing Machine/FB_HVAC_RND_Indoor_Unit.TcPOU
FUNCTION_BLOCK FB_HVAC_RND_Indoor_Unit EXTENDS FB_BaseDevice


VAR_INPUT
	nSetpoint: REAL; // This register stores indoor unit setpoint (0.1 degC step). This value multiplied by 10 to store as an integer value. 16bit signed integer
	nUnitID: STRING; //This will be set by the HVAC vendor - this is a DIINetID, and not a Modbus ID - do not confuse these?
					// The unit ID will be used to determine which bits to unpack from the modbus packets
					// The PLC will only receive Modbus messages from the centralised HVAC controller which has an individual Modbus ID
	
	// ----------------- Modbus Variables -----------//
	// Written in accordance with the modbus manuial supplied by vendor
	// https://drive.google.com/file/d/1Gl1Z8UXsnYqQFCh63b19Rq_Jpmyq9qef/view?usp=sharing
	
	// -------------------READ ONLY ---------------//

	// Status
	bConnectionStatus: BOOL;
	bCommsStatus: BOOL;

	// Status
	bOnOff_1_0: BOOL;
	
	nSetpoint_RO: REAL; // This register stores indoor unit setpoint (0.1 degC step). This value multiplied by 10 to store as an integer value. 16bit signed integer
	
	(*bForced: BOOL;
	nFanDirection_RO: UINT;
	nFanVolume_RO: UINT;
	nOperationMode_RO: UINT; // ENUM HERE?
	bFilterSignStatus: BOOL; // This comes through as a BYTE for all units, will need to access bit depending on the UNitID
	nOperationStatus_RO: UINT;
	nCoolHeatMaster: UINT;
	
	
	nErrorCode_Val1: UINT;
	nErrorCode_Val2: UINT;
	bMalfunction: BOOL;
	bWarning: BOOL;
	nRoomTemp: REAL; // This register stores indoor unit setpoint (0.1 degC step). This value multiplied by 10 to store as an integer value. 16bit signed integer
	bTempSensor_Error: BOOL;
	bTempSensor_DataReceived: BOOL;
	
	// -------------------READ / WRITE ---------------//
	(*
	
	nFanControlFlag: UINT;
	nFanDirection: UINT;
	nFanVolume: UINT;
	nOperationMode: UINT;
	nFilterSignReset: UINT;
	nOperationStatus: UINT; // Needs to be set before the cooling or heating setpoints are set
	*)
	*)
END_VAR

IF GVL.bAutoUpdateDeviceState THEN
	eState := eStateTarget;	
END_IF

IF NOT bConnectionStatus THEN
	raiseAlarm(Priority := E_AlarmPriority.High, Label := 'HVAC Indoor Unit Not Connected', Enabled := TRUE, DeviceAlarmID := 1);
ELSE
	raiseAlarm(Priority := E_AlarmPriority.High, Label := 'HVAC Indoor Unit Not Connected', Enabled := FALSE, DeviceAlarmID := 1);
END_IF

IF NOT bConnectionStatus THEN
	raiseAlarm(Priority := E_AlarmPriority.High, Label := 'HVAC Indoor Unit Comms Issue', Enabled := TRUE, DeviceAlarmID := 2);
ELSE
	raiseAlarm(Priority := E_AlarmPriority.High, Label := 'HVAC Indoor Unit Comms Issue', Enabled := FALSE, DeviceAlarmID := 2);
END_IF

END_FUNCTION_BLOCK

// ---- POUs/01 Actuators/Dosing Machine/FB_HVAC_RND_ModbusApadtor.TcPOU
FUNCTION_BLOCK FB_HVAC_RND_ModbusApadtor EXTENDS FB_BaseDevice

VAR
	
	// ----------------- Modbus Variables -----------//
	// Written in accordance with the modbus manuial supplied by vendor
	// https://drive.google.com/file/d/1Gl1Z8UXsnYqQFCh63b19Rq_Jpmyq9qef/view?usp=sharing
	
	// -------------------READ ONLY ---------------//
	bReady: BOOL;
	
	// -------------------READ / WRITE ---------------//
	bManagedDIINetAdr: BOOL;
	bDIINetMasterFlag: BOOL;
	bDIINet_Comms_StartStopFlag: BOOL;
	
	
	
END_VAR

END_FUNCTION_BLOCK

// ---- POUs/01 Actuators/Dosing Machine/FB_LevelWaterControl.TcPOU

(*
Function block to control opening and closing of water supply valve to the level
*)

{attribute 'OPC.UA.DA.StructuredType' := '1'}
FUNCTION_BLOCK FB_LevelWaterControl EXTENDS FB_BaseDevice
VAR_INPUT
	nStack : INT;
	nLevel : INT;
	
	bValve_NC_1_NO: BOOL;
	fbValve : FB_Valve_ONOFF_woMonitoring(ValveID := 'valveID' , ValveDescr := 'irrigation valve', Normal_State_NC_1_NO_0 := 0);
	{attribute 'OPC.UA.DA' := '1'}
	bActiveCropJob : BOOL;
	{attribute 'OPC.UA.DA' := '1'}
	tWaterOnTimer : TON;
	{attribute 'OPC.UA.DA' := '1'}
	tWaterOffTimer : TON;
	{attribute 'OPC.UA.DA' := '1'}
	tTimeTilWaterOff : TIME;
	{attribute 'OPC.UA.DA' := '1'}
	tTimeTilWaterOn : TIME;
	
	
	
END_VAR
VAR_OUTPUT
END_VAR
VAR
	{attribute 'OPC.UA.DA' := '1'}
	nMinutesOff : INT;
	{attribute 'OPC.UA.DA' := '1'}
	nMinutesOn : INT;
	{attribute 'OPC.UA.DA' := '1'}
	eValve_Mode : E_DeviceMode;
	{attribute 'OPC.UA.DA' := '1'}
	eValve_Command : E_DeviceState;
END_VAR


VAR_IN_OUT
	stSCInputs :ST_INPUTS_RND_StackControl;
END_VAR


// enable the water control. There is currently no way to Disable water control. Is there a use case for this?
// If you want to turn water off, you will have to put the valve into manual and close it.
//Inputs.LevelWaterControls[nLevel].bEnable := TRUE;

devicesUpdate();
waterTimers();
waterOnOff();
scanOPCinputs();

// stSCInputs.LevelWaterControls[nLevel].TimeUntilOn := TIME_TO_INT(tTimeTilWaterOn) / 1000;

METHOD devicesUpdate : BOOL
VAR_INPUT
END_VAR

//fbValve(bNO_or_NC_0_or_1 := stSCInputs.bIrrigValve_NC_1_NO_0);
fbValve();
END_METHOD

METHOD FB_init : BOOL
VAR_INPUT
	bInitRetains : BOOL; // if TRUE, the retain variables are initialized (warm start / cold start)
	bInCopyCode : BOOL;  // if TRUE, the instance afterwards gets moved into the copy code (online change)
END_VAR


// set the Water Control to Running. 
// There is currently no use case for the Water Control to be Stopped
eState := E_DeviceState.RUNNING;
END_METHOD

METHOD scanOPCinputs : BOOL
VAR_INPUT
END_VAR
fbValve.setMode(stSCInputs.LevelWaterControls[nLevel].Valve.Mode);

// set the valve's mode to the requested mode
IF NOT stSCInputs.bWaterQualityGood THEN            // inhibit irrigation if our water quality checkfromt the DM returns no bueno
	fbValve.close();
ELSE
	// OLD VERSION...fbValve.setMode(eValve_Mode);
	// NEW VERSION..
	
	
	IF fbValve.getMode() = E_DeviceMode.MANUAL THEN
		// the valve is in Manual so set the valve state to the input command
		IF stSCInputs.LevelWaterControls[nLevel].Valve.Command (*eValve_Command*) = E_DeviceState.OPEN THEN
			fbValve.open();
		END_IF
		IF stSCInputs.LevelWaterControls[nLevel].Valve.Command (*eValve_Command*) = E_DeviceState.CLOSED THEN
			fbValve.close();
		END_IF
	ELSE
		// the vale is not in Manual so set the Input command to the actual state
		// This prevents the valve from moving unexpectedly the next time someone puts it into Manual
		 stSCInputs.LevelWaterControls[nLevel].Valve.Command := fbValve.getState();
	END_IF
	
	
	IF stSCInputs.bParamsInitialised THEN
		nMinutesOn := stSCInputs.LevelWaterControls[1].MinutesOn;
		nMinutesOff := stSCInputs.LevelWaterControls[1].MinutesOff;
	END_IF

END_IF
END_METHOD

METHOD setState : BOOL
VAR_INPUT
	state : E_DeviceState;
END_VAR

eState := state;
END_METHOD

METHOD waterOnOff : BOOL
VAR_INPUT
END_VAR
IF fbValve.getMode() = E_DeviceMode.AUTO THEN
	IF bActiveCropJob THEN
		// crop movement is active on this level so turn the valve off
		fbValve.close();
	ELSIF eState <> E_DeviceState.RUNNING THEN
		// water is disabled on this level
		fbValve.close();
	ELSIF tWaterOnTimer.IN THEN
		fbValve.open();
	ELSE
		fbValve.close();
	END_IF
END_IF
END_METHOD

METHOD waterTimers : BOOL
VAR_INPUT
END_VAR

VAR
	tTimeOn : TIME;
	tTimeOff : TIME;
END_VAR
tTimeOff := DINT_TO_TIME(nMinutesOff * 60000);
tTimeOn := DINT_TO_TIME(nMinutesOn * 60000);

tWaterOnTimer(IN := nMinutesOn <> 0 AND 	(tWaterOffTimer.Q OR NOT tWaterOffTimer.IN), PT := tTimeOn); 
tWaterOffTimer(IN := nMinutesOff <> 0 AND 	(tWaterOnTimer.Q OR NOT tWaterOnTimer.IN), PT := tTimeOff); 


IF tWaterOffTimer.IN THEN
	tTimeTilWaterOff := T#0S;
	tTimeTilWaterOn := tWaterOffTimer.PT - tWaterOffTimer.ET;
ELSE
	tTimeTilWaterOn := T#0S;
	tTimeTilWaterOff := tWaterOnTimer.PT - tWaterOnTimer.ET;
END_IF
END_METHOD

END_FUNCTION_BLOCK

// ---- POUs/01 Actuators/Dosing Machine/FB_OxygenInjector.TcPOU
{attribute 'OPC.UA.DA.StructuredType' := '1'}
FUNCTION_BLOCK FB_OxygenInjector EXTENDS FB_BaseDevice IMPLEMENTS I_Device

VAR
	
	{attribute 'OPC.UA.DA' := '1'} 
	bInContactor AT %I*: BOOL := FALSE;
	{attribute 'OPC.UA.DA' := '1'} 
	bOutContactor AT %Q*: BOOL := FALSE;
	
	{attribute 'OPC.UA.DA' := '0'} 
	eSMState: (WAIT, TURNING_ON, ON, TURNING_OFF, OFF);
	
	{attribute 'OPC.UA.DA' := '0'} 
	tActionTimeout: TIME := T#5S;
	{attribute 'OPC.UA.DA' := '0'} 
	fbTON_timeout: TON := (PT := tActionTimeout, IN := FALSE);
END_VAR

fbTONstartTime();
fbTONstopTime();

IF GVL.bAutoUpdateDeviceState THEN
	eState := eStateTarget;	
END_IF

IF eMode = E_DeviceMode.AUTO AND (eStateTarget = E_DeviceState.ON) THEN
	bEnable := TRUE;
END_IF

IF eMode = E_DeviceMode.MANUAL THEN
	bEnable := TRUE;
END_IF

IF (bEnable AND (eStateTarget = E_DeviceState.ON)) AND eSMState <> ON THEN
		eSMState := TURNING_ON;
END_IF

IF ((bEnable = FALSE) OR (eStateTarget = E_DeviceState.OFF)) AND eSMState <> OFF THEN
		eSMState := TURNING_OFF;
END_IF



CASE eSMState OF
	
	WAIT:
		//Wait for method call to change ESMState
		eState := E_DeviceState.OFF;
		bOutContactor := FALSE;
		
	TURNING_ON: 
		eState := E_DeviceState.TURNING_ON;
		eSMState := ON;
		bOutContactor := TRUE;
	
	ON:
		eState := E_DeviceState.ON;
		bOutContactor := TRUE;
		
		
	TURNING_OFF:

		bOutContactor := FALSE;
		eSMState := OFF;
		
		
	OFF:
		eState := E_DeviceState.OFF;
		bOutContactor := FALSE;
		
END_CASE

{warning 'add method implementation '}
METHOD disable : BOOL
bEnable := FALSE;
END_METHOD

{warning 'add method implementation '}
METHOD enable : BOOL
bEnable := TRUE;
END_METHOD

METHOD FB_init : BOOL
VAR_INPUT
	bInitRetains : BOOL; // if TRUE, the retain variables are initialized (warm start / cold start)
	bInCopyCode : BOOL;  // if TRUE, the instance afterwards gets moved into the copy code (online change)
	
	UnitID: STRING(80);
	UnitDescr: STRING(255); 
END_VAR
sID := UnitID;
sDescr := UnitDescr;
END_METHOD

METHOD setOff : BOOL
VAR_INPUT
END_VAR
eStateTarget := E_DeviceState.OFF;
END_METHOD

METHOD setOn : BOOL
VAR_INPUT
END_VAR
eStateTarget := E_DeviceState.ON;
END_METHOD

END_FUNCTION_BLOCK

// ---- POUs/01 Actuators/Dosing Machine/FB_OxygenInjector_1.TcPOU
{attribute 'OPC.UA.DA.StructuredType' := '1'}
FUNCTION_BLOCK FB_OxygenInjector_1 EXTENDS FB_BaseDevice IMPLEMENTS I_Device

VAR
	
	{attribute 'OPC.UA.DA' := '1'} 
	bInContactor AT %I*: BOOL := FALSE;
	{attribute 'OPC.UA.DA' := '1'} 
	bOutContactor AT %Q*: BOOL := FALSE;
	
	{attribute 'OPC.UA.DA' := '0'} 
	eSMState: (WAIT, TURNING_ON, ON, TURNING_OFF, OFF);
	
	{attribute 'OPC.UA.DA' := '0'} 
	tActionTimeout: TIME := T#5S;
	{attribute 'OPC.UA.DA' := '0'} 
	fbTON_timeout: TON := (PT := tActionTimeout, IN := FALSE);
END_VAR

fbTONstartTime();
fbTONstopTime();

IF GVL.bAutoUpdateDeviceState THEN
	eState := eStateTarget;	
END_IF


IF eMode = E_DeviceMode.MANUAL THEN
	bEnable := TRUE;
END_IF

IF bEnable AND eStateTarget = E_DeviceState.ON AND eState <> E_DeviceState.ON THEN
		eSMState := TURNING_ON;
END_IF

IF bEnable = FALSE OR (eStateTarget = E_DeviceState.OFF AND eState <> E_DeviceState.OFF) THEN
		eSMState := TURNING_OFF;
END_IF


CASE eSMState OF
	
	WAIT:
		//Wait for method call to change ESMState
		
	TURNING_ON: 
		eState := E_DeviceState.TURNING_ON;

		bOutContactor := TRUE;
	
		IF fbTONstartTime.Q THEN
			eSMState := WAIT;
			raiseAlarm(Priority := E_AlarmPriority.High, Label := 'Failed to Start', Enabled := TRUE, DeviceAlarmID := 1);
		END_IF
		
		IF bInContactor  THEN
			eSMState := ON;
			eState := E_DeviceState.ON;
		END_IF
		
	ON:
		IF bInContactor <> TRUE THEN
			raiseAlarm(Priority := E_AlarmPriority.High, Label := 'Power Lost', Enabled := TRUE, DeviceAlarmID := 2);
			eState := E_DeviceState.OFF;
			eSMState := WAIT;
		END_IF
		

		
	TURNING_OFF:
		eState := E_DeviceState.TURNING_OFF;
		bOutContactor := FALSE;

				
		IF fbTONstopTime.Q THEN
			eSMState := WAIT;
			raiseAlarm(Priority := E_AlarmPriority.High, Label := 'Failed to Stop', Enabled := TRUE, DeviceAlarmID := 3);
		END_IF 
		
		IF bInContactor = FALSE THEN
			eSMState := OFF;	
		END_IF
		

	OFF:
		eState := E_DeviceState.OFF;
		eSMState := WAIT;
		
		
END_CASE

{warning 'add method implementation '}
METHOD disable : BOOL
bEnable := FALSE;
END_METHOD

{warning 'add method implementation '}
METHOD enable : BOOL
bEnable := TRUE;
END_METHOD

METHOD FB_init : BOOL
VAR_INPUT
	bInitRetains : BOOL; // if TRUE, the retain variables are initialized (warm start / cold start)
	bInCopyCode : BOOL;  // if TRUE, the instance afterwards gets moved into the copy code (online change)
	
	UnitID: STRING(80);
	UnitDescr: STRING(255); 
END_VAR
sID := UnitID;
sDescr := UnitDescr;
END_METHOD

METHOD setOff : BOOL
VAR_INPUT
END_VAR
eSMState := TURNING_OFF;
END_METHOD

METHOD setOn : BOOL
VAR_INPUT
END_VAR
eSMState := TURNING_ON;
END_METHOD

END_FUNCTION_BLOCK

// ---- POUs/01 Actuators/Dosing Machine/FB_OzoneGenerator.TcPOU
{attribute 'OPC.UA.DA.StructuredType' := '1'}
FUNCTION_BLOCK FB_OzoneGenerator EXTENDS FB_BaseDevice IMPLEMENTS I_Device

VAR
	{attribute 'OPC.UA.DA' := '1'} 
	bInContactor AT %I*: BOOL := FALSE;
	{attribute 'OPC.UA.DA' := '1'} 
	bOutContactor AT %Q*: BOOL := FALSE;
	
	{attribute 'OPC.UA.DA' := '0'} 
	eSMState: (WAIT, TURNING_ON, ON, TURNING_OFF, OFF);
	
	{attribute 'OPC.UA.DA' := '0'} 
	tActionTimeout: TIME := T#5S;
	{attribute 'OPC.UA.DA' := '0'} 
	fbTON_timeout: TON := (PT := tActionTimeout, IN := FALSE);
END_VAR

fbTONstartTime();
fbTONstopTime();

IF GVL.bAutoUpdateDeviceState THEN
	eState := eStateTarget;	
END_IF


IF bEnable THEN
	IF eStateTarget = E_DeviceState.ON AND eState <> E_DeviceState.ON THEN
		eSMState := TURNING_ON;
	END_IF
END_IF

IF eStateTarget = E_DeviceState.OFF AND eState <> E_DeviceState.OFF THEN
		eSMState := TURNING_OFF;
END_IF


CASE eSMState OF
	
	WAIT:
		//Wait for method call to change ESMState
		
	TURNING_ON: 
		eState := E_DeviceState.TURNING_ON;

		bOutContactor := TRUE;
	
		IF fbTONstartTime.Q THEN
			eSMState := WAIT;
			raiseAlarm(Priority := E_AlarmPriority.High, Label := 'Failed to Start', Enabled := TRUE, DeviceAlarmID := 1);
		END_IF
		
		IF bInContactor  THEN
			eSMState := ON;
			eState := E_DeviceState.ON;
		END_IF
		
	ON:
		IF bInContactor <> TRUE THEN
			raiseAlarm(Priority := E_AlarmPriority.High, Label := 'Power Lost', Enabled := TRUE, DeviceAlarmID := 2);
			eState := E_DeviceState.OFF;
			eSMState := WAIT;
		END_IF
		

		
	TURNING_OFF:
		eState := E_DeviceState.TURNING_OFF;
		bOutContactor := FALSE;

				
		IF fbTONstopTime.Q THEN
			eSMState := WAIT;
			raiseAlarm(Priority := E_AlarmPriority.High, Label := 'Failed to Stop', Enabled := TRUE, DeviceAlarmID := 3);
		END_IF 
		
		IF bInContactor = FALSE THEN
			eSMState := OFF;	
		END_IF
		

	OFF:
		eState := E_DeviceState.OFF;
		eSMState := WAIT;
		
		
END_CASE

{warning 'add method implementation '}
METHOD disable : BOOL
bEnable := FALSE;
END_METHOD

{warning 'add method implementation '}
METHOD enable : BOOL
bEnable := TRUE;
END_METHOD

METHOD FB_init : BOOL
VAR_INPUT
	bInitRetains : BOOL; // if TRUE, the retain variables are initialized (warm start / cold start)
	bInCopyCode : BOOL;  // if TRUE, the instance afterwards gets moved into the copy code (online change)
	
	UnitID: STRING(80);
	UnitDescr: STRING(255); 
END_VAR
sID := UnitID;
sDescr := UnitDescr;
END_METHOD

METHOD setOff : BOOL
VAR_INPUT
END_VAR
eSMState := TURNING_OFF;
END_METHOD

METHOD setOn : BOOL
VAR_INPUT
END_VAR
eSMState := TURNING_ON;
END_METHOD

END_FUNCTION_BLOCK

// ---- POUs/01 Actuators/Dosing Machine/FB_PumpDOL_Onga413.TcPOU
{attribute 'OPC.UA.DA.StructuredType' := '1'}
FUNCTION_BLOCK FB_PumpDOL_Onga413 EXTENDS FB_BaseDevice IMPLEMENTS I_Device, I_PumpVSD

VAR
	{attribute 'OPC.UA.DA' := '1'} 
	bInContactor AT %I*: BOOL := FALSE;
	{attribute 'OPC.UA.DA' := '1'} 
	bOutContactor AT %Q*: BOOL := FALSE;


	//MB:  REFERENCE TO FB_ModbusMaster;
	{attribute 'OPC.UA.DA' := '1'} 
	nFrequencySetPoint: REAL := 0;
	{attribute 'OPC.UA.DA' := '1'} 
	nFrequencyActual: REAL := 0;
	
	{attribute 'OPC.UA.DA' := '0'} 
	eSMState: (WAIT, STARTING, RUNNING, STOPPING, STOPPED);
	
END_VAR

fbTONstartTime();
fbTONstopTime();

IF GVL.bAutoUpdateDeviceState THEN
	eState := eStateTarget;	
END_IF



IF bEnable THEN
	IF eStateTarget = E_DeviceState.ON AND eState <> E_DeviceState.ON THEN
		eSMState := STARTING;
	END_IF
END_IF

IF eStateTarget = E_DeviceState.OFF AND eState <> E_DeviceState.OFF THEN
		eSMState := STOPPING;
END_IF


CASE eSMState OF
	
	WAIT:
		//Wait for method call to change ESMState
		
	STARTING: 
		eState := E_DeviceState.STARTING;

		bOutContactor := TRUE;
	
		IF fbTONstartTime.Q THEN
			eSMState := WAIT;
			raiseAlarm(Priority := E_AlarmPriority.High, Label := 'Failed to Start', Enabled := TRUE, DeviceAlarmID := 2);
		END_IF
		
		IF bInContactor THEN
			eSMState := RUNNING;
			eState := E_DeviceState.RUNNING;
		END_IF
		
	RUNNING:
		IF bInContactor <> TRUE THEN
			raiseAlarm(Priority := E_AlarmPriority.High, Label := 'Power Lost', Enabled := TRUE, DeviceAlarmID := 2);
			eState := E_DeviceState.FAULTED;
			eSMState := WAIT;
		END_IF
		
		// Add pump / motor control here - look at built in Twincat libraries 
		// Add relevant VSD signals to check
		

	STOPPING:
		eState := E_DeviceState.STOPPING;
		bOutContactor := FALSE;
				
		IF fbTONstopTime.Q THEN
			eSMState := WAIT;
			raiseAlarm(Priority := E_AlarmPriority.High, Label := 'Failed to Stop', Enabled := TRUE, DeviceAlarmID := 3);
		END_IF 
		
		IF bInContactor = FALSE AND nFrequencyActual = 0 THEN
			eSMState := STOPPED;	
		END_IF
		

	STOPPED:
		eState := E_DeviceState.IDLE;
		eSMState := WAIT;
		
		
END_CASE

{warning 'add method implementation '}
METHOD disable : BOOL
END_METHOD

{warning 'add method implementation '}
METHOD enable : BOOL
END_METHOD

{warning 'add method implementation '}
METHOD FB_init : BOOL
VAR_INPUT
	(* if TRUE, the retain variables are initialized (warm start / cold start)*)
	bInitRetains	: BOOL;
	(* if TRUE, the instance afterwards gets moved into the copy code (online change)*)
	bInCopyCode	: BOOL;
	PumpID	: STRING(80);
	PumpDescr	: STRING(255);
END_VAR
sID := PumpID;
sDescr := PumpDescr;
END_METHOD

{warning 'add method implementation '}
METHOD getFrequency : REAL
END_METHOD

METHOD setModbusMaster : BOOL
METHOD setModbusMaster : BOOL
VAR_INPUT
	//ModbusMaster: REFERENCE TO FB_ModbusMaster;
END_VAR
//MB := ModbusMaster;
END_METHOD

METHOD setOff : BOOL
VAR_INPUT
END_VAR
END_METHOD

METHOD setOn : BOOL
VAR_INPUT
END_VAR
END_METHOD

{warning 'add method implementation '}
METHOD setReference : BOOL
VAR_INPUT
	RefSetPoint	: REAL;
END_VAR
END_METHOD

END_FUNCTION_BLOCK

// ---- POUs/01 Actuators/Dosing Machine/FB_PumpDOL_Onga413_RND.TcPOU
{attribute 'OPC.UA.DA.StructuredType' := '1'}
FUNCTION_BLOCK FB_PumpDOL_Onga413_RND EXTENDS FB_BaseDevice IMPLEMENTS I_Device, I_PumpVSD

VAR
	bFirstRun: BOOL := TRUE;
	{attribute 'OPC.UA.DA' := '1'} 
	bInContactor AT %I*: BOOL := FALSE;
	{attribute 'OPC.UA.DA' := '1'} 
	bOutContactor AT %Q*: BOOL := FALSE;

	
	fbTON_OnTimer: TON := (PT := tTimeOn, IN := FALSE);
	tTimeOn: TIME := T#15S;
	
	//MB:  REFERENCE TO FB_ModbusMaster;
	{attribute 'OPC.UA.DA' := '1'}
	nFrequencySetPoint: REAL := 0;
	{attribute 'OPC.UA.DA' := '1'}
	nFrequencyActual: REAL := 0;
	
	{attribute 'OPC.UA.DA' := '0'} 
	eSMState: (WAIT, STARTING, RUNNING, STOPPING, STOPPED);
	
	tDebounce: TIME := T#5S;
	fbTON_Debounce: TON := (PT := tDebounce, IN := FALSE);
	
END_VAR

IF bFirstRun THEN
	bFirstRun := FALSE;

END_IF

fbTON_Debounce();
fbTONstartTime(PT := tTimeOn);
fbTON_OnTimer(PT := tTimeOn);
fbTONstopTime();



IF GVL.bAutoUpdateDeviceState THEN
	eState := eStateTarget;	
END_IF




IF eMode = E_DeviceMode.MANUAL THEN
	bEnable := TRUE;
END_IF

IF bEnable AND (eStateTarget = E_DeviceState.RUNNING) AND eSMState <> RUNNING THEN
		eSMState := STARTING;
		fbTON_Debounce(IN := TRUE);
		fbTON_OnTimer(IN := TRUE);
		
END_IF

IF (bEnable = FALSE OR eStateTarget = E_DeviceState.IDLE) AND eSMState <> WAIT THEN
		eSMState := STOPPING;
		fbTON_Debounce(IN := FALSE);
		fbTON_OnTimer(IN := FALSE);
END_IF


(*

CASE eSMState OF
	
	WAIT:
		//Wait for method call to change ESMState
		fbTON_OnTimer(IN := FALSE);
		
	STARTING: 
	
		IF fbTON_Debounce.Q THEN
			eState := E_DeviceState.STARTING;
			fbTON_OnTimer(IN := TRUE);
			bOutContactor := TRUE;
		
			IF fbTONstartTime.Q THEN
				eSMState := WAIT;
				raiseAlarm(Priority := E_AlarmPriority.High, Label := 'Failed to Start', Enabled := TRUE, DeviceAlarmID := 1);
			END_IF
			
			IF TRUE THEN
				eSMState := RUNNING;
				eState := E_DeviceState.RUNNING;
			END_IF
			fbTON_Debounce(IN := FALSE);
		END_IF

		
	RUNNING:
		IF bOutContactor <> TRUE THEN
			raiseAlarm(Priority := E_AlarmPriority.High, Label := 'Power Lost', Enabled := TRUE, DeviceAlarmID := 2);
			eState := E_DeviceState.IDLE;
			eSMState := WAIT;
		END_IF
		
		// Add pump / motor control here - look at built in Twincat libraries 
		// Add relevant VSD signals to check
		

	STOPPING:
		eState := E_DeviceState.STOPPING;
		bOutContactor := FALSE;
		eSMState := STOPPED;

		

	STOPPED:
		eState := E_DeviceState.IDLE;
		fbTON_Debounce(IN := TRUE);
		eSMState := WAIT;
		
		
END_CASE

*)

CASE eSMState OF
	
	WAIT:
		//Wait for method call to change ESMState
		
	STARTING: 
		IF fbTON_Debounce.Q THEN
			eState := E_DeviceState.STARTING;
			bOutContactor := TRUE;
			fbTON_Debounce.IN := FALSE;
			eSMState := RUNNING;
		END_IF

		
	RUNNING:
		eState := E_DeviceState.RUNNING;
		IF bOutContactor <> TRUE THEN
			raiseAlarm(Priority := E_AlarmPriority.High, Label := 'Power Lost', Enabled := TRUE, DeviceAlarmID := 1);
			eSMState := STOPPING;
		END_IF
			
	STOPPING:
		fbTON_Debounce.IN := TRUE;
		fbTON_OnTimer(IN := FALSE);
		bOutContactor := TRUE;
		eState := E_DeviceState.STOPPING;
		bOutContactor := FALSE;
		eSMState := STOPPED;

	STOPPED:
		eState := E_DeviceState.IDLE;
		eSMState := WAIT;
		fbTON_Debounce.IN := TRUE;
		
END_CASE

{warning 'add method implementation '}
METHOD disable : BOOL
bEnable := FALSE;
END_METHOD

{warning 'add method implementation '}
METHOD enable : BOOL
bEnable := TRUE;
END_METHOD

{warning 'add method implementation '}
METHOD FB_init : BOOL
VAR_INPUT
	(* if TRUE, the retain variables are initialized (warm start / cold start)*)
	bInitRetains	: BOOL;
	(* if TRUE, the instance afterwards gets moved into the copy code (online change)*)
	bInCopyCode	: BOOL;
	PumpID	: STRING(80);
	PumpDescr	: STRING(255);
END_VAR
sID := PumpID;
sDescr := PumpDescr;
END_METHOD

{warning 'add method implementation '}
METHOD getFrequency : REAL
END_METHOD

METHOD setModbusMaster : BOOL
METHOD setModbusMaster : BOOL
VAR_INPUT
	//ModbusMaster: REFERENCE TO FB_ModbusMaster;
END_VAR
//MB := ModbusMaster;
END_METHOD

METHOD setOff : BOOL
VAR_INPUT
END_VAR
END_METHOD

METHOD setOn : BOOL
VAR_INPUT
END_VAR
END_METHOD

{warning 'add method implementation '}
METHOD setReference : BOOL
VAR_INPUT
	RefSetPoint	: REAL;
END_VAR
END_METHOD

METHOD startTimer : BOOL
VAR_INPUT
END_VAR
startTimer := fbTON_OnTimer.Q;
END_METHOD

END_FUNCTION_BLOCK

// ---- POUs/01 Actuators/Dosing Machine/FB_PumpVSD_DanfossFC202.TcPOU
{attribute 'OPC.UA.DA.StructuredType' := '1'}
FUNCTION_BLOCK FB_PumpVSD_DanfossFC202 EXTENDS FB_BaseDevice IMPLEMENTS I_Device, I_PumpVSD

VAR
	{attribute 'OPC.UA.DA' := '0'} 
	bInContactor AT %I*: BOOL := FALSE;
	{attribute 'OPC.UA.DA' := '0'} 
	bOutContactor AT %Q*: BOOL := FALSE;

	//MB:  REFERENCE TO FB_ModbusMaster;
	{attribute 'OPC.UA.DA' := '1'} 
	nFrequencySetPoint: REAL := 0;
	{attribute 'OPC.UA.DA' := '1'}
	nFrequencyActual: REAL := 0;
	
	{attribute 'OPC.UA.DA' := '0'} 
	eSMState: (WAIT, STARTING, RUNNING, STOPPING, STOPPED);
	
END_VAR

fbTONstartTime();
fbTONstopTime();

IF GVL.bAutoUpdateDeviceState THEN
	eState := eStateTarget;	
END_IF



IF bEnable THEN
	IF eStateTarget = E_DeviceState.ON AND eState <> E_DeviceState.ON THEN
		eSMState := STARTING;
	END_IF
END_IF

IF eStateTarget = E_DeviceState.OFF AND eState <> E_DeviceState.OFF THEN
		eSMState := STOPPING;
END_IF


CASE eSMState OF
	
	WAIT:
		//Wait for method call to change ESMState
		
	STARTING: 
		eState := E_DeviceState.STARTING;

		bOutContactor := TRUE;
	
		IF fbTONstartTime.Q THEN
			eSMState := WAIT;
			raiseAlarm(Priority := E_AlarmPriority.High, Label := 'Failed to Start', Enabled := TRUE, DeviceAlarmID := 1);
		END_IF
		
		IF bInContactor THEN
			eSMState := RUNNING;
			eState := E_DeviceState.ON;
		END_IF
		
	RUNNING:
		IF bInContactor <> TRUE THEN
			raiseAlarm(Priority := E_AlarmPriority.High, Label := 'Power Lost', Enabled := TRUE, DeviceAlarmID := 2);
			eState := E_DeviceState.OFF;
			eSMState := WAIT;
		END_IF
		
		// Add pump / motor control here - look at built in Twincat libraries 
		// Add relevant VSD signals to check
		

	STOPPING:
		eState := E_DeviceState.STOPPING;
		bOutContactor := FALSE;
				
		IF fbTONstopTime.Q THEN
			eSMState := WAIT;
			raiseAlarm(Priority := E_AlarmPriority.High, Label := 'Failed to Stop', Enabled := TRUE, DeviceAlarmID := 3);
		END_IF 
		
		IF bInContactor = FALSE AND nFrequencyActual = 0 THEN
			eSMState := STOPPED;	
		END_IF
		

	STOPPED:
		eState := E_DeviceState.IDLE;
		eSMState := WAIT;
		
		
END_CASE

{warning 'add method implementation '}
METHOD disable : BOOL
END_METHOD

{warning 'add method implementation '}
METHOD enable : BOOL
END_METHOD

{warning 'add method implementation '}
METHOD FB_init : BOOL
VAR_INPUT
	(* if TRUE, the retain variables are initialized (warm start / cold start)*)
	bInitRetains	: BOOL;
	(* if TRUE, the instance afterwards gets moved into the copy code (online change)*)
	bInCopyCode	: BOOL;
	PumpID	: STRING(80);
	PumpDescr	: STRING(255);
END_VAR
sID := PumpID;
sDescr := PumpDescr;
END_METHOD

{warning 'add method implementation '}
METHOD getFrequency : REAL
END_METHOD

METHOD setModbusMaster : BOOL
METHOD setModbusMaster : BOOL
VAR_INPUT
	//ModbusMaster: REFERENCE TO FB_ModbusMaster;
END_VAR
//MB := ModbusMaster;
END_METHOD

METHOD setOff : BOOL
VAR_INPUT
END_VAR
END_METHOD

METHOD setOn : BOOL
VAR_INPUT
END_VAR
END_METHOD

{warning 'add method implementation '}
METHOD setReference : BOOL
VAR_INPUT
	RefSetPoint	: REAL;
END_VAR
END_METHOD

END_FUNCTION_BLOCK

// ---- POUs/01 Actuators/Dosing Machine/FB_PumpVSD_GrundfosCUE.TcPOU
{attribute 'OPC.UA.DA.StructuredType' := '1'}
FUNCTION_BLOCK FB_PumpVSD_GrundfosCUE EXTENDS FB_BaseDevice IMPLEMENTS I_Device, I_PumpVSD

VAR_IN_OUT
	{attribute 'OPC.UA.DA' := '0'}
	fbModbusMaster: FB_ModbusMaster;
END_VAR


VAR

	//MB:  REFERENCE TO FB_ModbusMaster;
	{attribute 'OPC.UA.DA' := '1'} 
	bInContactor AT %I*: BOOL := FALSE;
	{attribute 'OPC.UA.DA' := '1'} 
	bOutContactor AT %Q*: BOOL := FALSE;
	
	{attribute 'OPC.UA.DA' := '1'} 
	nFrequencySetPoint: REAL := 0;
	{attribute 'OPC.UA.DA' := '1'} 
	nFrequencyActual: REAL := 0;
	
	{attribute 'OPC.UA.DA' := '0'} 
	eSMState: (WAIT, STARTING, RUNNING, STOPPING, STOPPED);
	
END_VAR

fbTONstartTime();
fbTONstopTime();

IF GVL.bAutoUpdateDeviceState THEN
	eState := eStateTarget;	
END_IF


IF bEnable THEN
	IF eStateTarget = E_DeviceState.ON AND eState <> E_DeviceState.ON THEN
		eSMState := STARTING;
	END_IF
END_IF

IF eStateTarget = E_DeviceState.OFF AND eState <> E_DeviceState.OFF THEN
		eSMState := STOPPING;
END_IF


CASE eSMState OF
	
	WAIT:
		//Wait for method call to change ESMState
		
	STARTING: 
		eState := E_DeviceState.STARTING;

		bOutContactor := TRUE;
	
		IF fbTONstartTime.Q THEN
			eSMState := WAIT;
			raiseAlarm(Priority := E_AlarmPriority.High, Label := 'Failed to Start', Enabled := TRUE, DeviceAlarmID := 1);
		END_IF
		
		IF bInContactor THEN
			eSMState := RUNNING;
			eState := E_DeviceState.ON;
		END_IF
		
	RUNNING:
		IF bInContactor <> TRUE THEN
			raiseAlarm(Priority := E_AlarmPriority.High, Label := 'Power Lost', Enabled := TRUE, DeviceAlarmID := 2);
			eState := E_DeviceState.OFF;
			eSMState := WAIT;
		END_IF
		
		// Add pump / motor control here - look at built in Twincat libraries 
		// Add relevant VSD signals to check
		

	STOPPING:
		eState := E_DeviceState.STOPPING;
		bOutContactor := FALSE;
				
		IF fbTONstopTime.Q THEN
			eSMState := WAIT;
			raiseAlarm(Priority := E_AlarmPriority.High, Label := 'Failed to Stop', Enabled := TRUE, DeviceAlarmID := 3);
		END_IF 
		
		IF bInContactor = FALSE AND nFrequencyActual = 0 THEN
			eSMState := STOPPED;	
		END_IF
		

	STOPPED:
		eState := E_DeviceState.IDLE;
		eSMState := WAIT;
		
		
END_CASE

{warning 'add method implementation '}
METHOD disable : BOOL
END_METHOD

{warning 'add method implementation '}
METHOD enable : BOOL
END_METHOD

{warning 'add method implementation '}
METHOD FB_init : BOOL
VAR_INPUT
	(* if TRUE, the retain variables are initialized (warm start / cold start)*)
	bInitRetains	: BOOL;
	(* if TRUE, the instance afterwards gets moved into the copy code (online change)*)
	bInCopyCode	: BOOL;
	PumpID	: STRING(80);
	PumpDescr	: STRING(255);
END_VAR
sID := PumpID;
sDescr := PumpDescr;
END_METHOD

{warning 'add method implementation '}
METHOD getFrequency : REAL
END_METHOD

METHOD setModbusMaster : BOOL
METHOD setModbusMaster : BOOL
VAR_INPUT
	//ModbusMaster: REFERENCE TO FB_ModbusMaster;
END_VAR
//MB := ModbusMaster;
END_METHOD

METHOD setOff : BOOL
VAR_INPUT
END_VAR
END_METHOD

METHOD setOn : BOOL
VAR_INPUT
END_VAR
END_METHOD

{warning 'add method implementation '}
METHOD setReference : BOOL
VAR_INPUT
	RefSetPoint	: REAL;
END_VAR
END_METHOD

END_FUNCTION_BLOCK

// ---- POUs/01 Actuators/Dosing Machine/FB_UltraSonicCleaner.TcPOU
{attribute 'OPC.UA.DA.StructuredType' := '1'}
FUNCTION_BLOCK FB_UltraSonicCleaner EXTENDS FB_BaseDevice IMPLEMENTS I_Device

VAR
	{attribute 'OPC.UA.DA' := '1'} 
	bInContactor AT %I*: BOOL := FALSE;
	{attribute 'OPC.UA.DA' := '1'} 
	bOutContactor AT %Q*: BOOL := FALSE;
	
	{attribute 'OPC.UA.DA' := '0'} 
	eSMState: (WAIT, TURNING_ON, ON, TURNING_OFF, OFF);
	
	{attribute 'OPC.UA.DA' := '0'} 
	tActionTimeout: TIME := T#5S;
	{attribute 'OPC.UA.DA' := '0'} 
	fbTON_timeout: TON := (PT := tActionTimeout, IN := FALSE);
END_VAR

fbTONstartTime();
fbTONstopTime();

IF GVL.bAutoUpdateDeviceState THEN
	eState := eStateTarget;	
END_IF


IF bEnable THEN
	IF eStateTarget = E_DeviceState.ON AND eState <> E_DeviceState.ON THEN
		eSMState := TURNING_ON;
	END_IF
END_IF

IF eStateTarget = E_DeviceState.OFF AND eState <> E_DeviceState.OFF THEN
		eSMState := TURNING_OFF;
END_IF



CASE eSMState OF
	
	WAIT:
		//Wait for method call to change ESMState
		
	TURNING_ON: 
		bOutContactor := TRUE;
		eSMState := ON;
		eState := E_DeviceState.TURNING_ON;
		
		IF fbTONstartTime.Q THEN
			eSMState := WAIT;
			raiseAlarm(Priority := E_AlarmPriority.High, Label := 'Drum Filter Failed to Start', Enabled := TRUE, DeviceAlarmID := 1);
		END_IF
		
		
	ON:
		IF bInContactor = TRUE THEN
			eState := E_DeviceState.ON;
			eSMState := WAIT;
			bBusy := FALSE;
		END_IF	
	
		
	TURNING_OFF:
		bOutContactor := FALSE;
		eSMState := OFF;
		eState := E_DeviceState.TURNING_OFF;
		
		IF fbTONstopTime.Q THEN
			eSMState := WAIT;
			raiseAlarm(Priority := E_AlarmPriority.High, Label := 'Drum Filter Failed to Stop', Enabled := TRUE, DeviceAlarmID := 2);
		END_IF 
		

	OFF:
		IF bInContactor = FALSE THEN
			eState := E_DeviceState.OFF;
			eSMState := WAIT;
			bBusy := FALSE;
		END_IF
END_CASE

{warning 'add method implementation '}
METHOD disable : BOOL
bEnable := FALSE;
END_METHOD

{warning 'add method implementation '}
METHOD enable : BOOL
bEnable := TRUE;
END_METHOD

METHOD FB_init : BOOL
VAR_INPUT
	bInitRetains : BOOL; // if TRUE, the retain variables are initialized (warm start / cold start)
	bInCopyCode : BOOL;  // if TRUE, the instance afterwards gets moved into the copy code (online change)
	
	UnitID: STRING(80);
	UnitDescr: STRING(255); 
END_VAR
sID := UnitID;
sDescr := UnitDescr;
END_METHOD

METHOD setOff : BOOL
VAR_INPUT
END_VAR
eSMState := TURNING_OFF;
END_METHOD

METHOD setOn : BOOL
VAR_INPUT
END_VAR
eSMState := TURNING_ON;
END_METHOD

END_FUNCTION_BLOCK

// ---- POUs/01 Actuators/Dosing Machine/FB_Unit_RO_PW30_1.TcPOU
{attribute 'OPC.UA.DA.StructuredType' := '1'}
FUNCTION_BLOCK FB_Unit_RO_PW30_1 EXTENDS FB_BaseDevice IMPLEMENTS I_Device

VAR
	{attribute 'OPC.UA.DA' := '1'} 
	bInContactor AT %I*: BOOL := FALSE;
	{attribute 'OPC.UA.DA' := '1'} 
	bInRun AT %I*: BOOL := FALSE;
	{attribute 'OPC.UA.DA' := '1'} 
	bInAlarm AT %I*: BOOL := FALSE;
	
	{attribute 'OPC.UA.DA' := '1'} 
	bOutContactor AT %Q*: BOOL := FALSE;
	{attribute 'OPC.UA.DA' := '1'} 
	bOutON AT %Q*: BOOL := FALSE;
	{attribute 'OPC.UA.DA' := '1'} 
	bOutEnable AT %Q*: BOOL := FALSE;
	
	{attribute 'OPC.UA.DA' := '0'} 
	eSMState: (WAIT, TURNING_ON, ON, TURNING_OFF, OFF);
	
	{attribute 'OPC.UA.DA' := '0'} 
	tActionTimeout: TIME := T#5S;
	{attribute 'OPC.UA.DA' := '0'} 
	fbTON_timeout: TON := (PT := tActionTimeout, IN := FALSE);
END_VAR

fbTONstartTime();
fbTONstopTime();

IF GVL.bAutoUpdateDeviceState THEN
	eState := eStateTarget;	
END_IF


IF bEnable THEN
	IF eStateTarget = E_DeviceState.ON AND eState <> E_DeviceState.ON THEN
		eSMState := TURNING_ON;
	END_IF
END_IF

IF eStateTarget = E_DeviceState.OFF AND eState <> E_DeviceState.OFF THEN
		eSMState := TURNING_OFF;
END_IF

IF bInAlarm THEN
	raiseAlarm(Priority := E_AlarmPriority.High, Label := 'Unit Alarm Active', Enabled := TRUE, DeviceAlarmID := 1);
END_IF


CASE eSMState OF
	
	WAIT:
		//Wait for method call to change ESMState
		
	TURNING_ON: 
		eState := E_DeviceState.TURNING_ON;
		
		bOutContactor := TRUE;
		bOutEnable := TRUE;
		bOutON := TRUE;
	
		
		IF fbTONstartTime.Q THEN
			eSMState := WAIT;
			raiseAlarm(Priority := E_AlarmPriority.High, Label := 'Failed to Start', Enabled := TRUE, DeviceAlarmID := 2);
		END_IF
		
		IF bInContactor AND bInRun THEN
			eSMState := ON;
			eState := E_DeviceState.ON;
		END_IF
		
	ON:
		IF bInContactor <> TRUE THEN
			raiseAlarm(Priority := E_AlarmPriority.High, Label := 'Power Lost', Enabled := TRUE, DeviceAlarmID := 1);
			eState := E_DeviceState.OFF;
			eSMState := WAIT;
		END_IF
		
		IF bInRun <> TRUE THEN
			raiseAlarm(Priority := E_AlarmPriority.High, Label := 'Unit Stopped Running', Enabled := TRUE, DeviceAlarmID := 2);
			eState := E_DeviceState.OFF;
			eSMState := WAIT;
		END_IF
			
		
	TURNING_OFF:
		eState := E_DeviceState.TURNING_OFF;
		bOutContactor := FALSE;
		bOutON := FALSE;
		bOutEnable := FALSE;
				
		IF fbTONstopTime.Q THEN
			eSMState := WAIT;
			raiseAlarm(Priority := E_AlarmPriority.High, Label := 'Failed to Stop', Enabled := TRUE, DeviceAlarmID := 3);
		END_IF 
		
		IF bInRun = FALSE AND bInContactor = FALSE THEN
			eSMState := OFF;	
		END_IF
		

	OFF:
		eState := E_DeviceState.OFF;
		eSMState := WAIT;
		
		
END_CASE

{warning 'add method implementation '}
METHOD disable : BOOL
bEnable := FALSE;
END_METHOD

{warning 'add method implementation '}
METHOD enable : BOOL
bEnable := TRUE;
END_METHOD

METHOD FB_init : BOOL
VAR_INPUT
	bInitRetains : BOOL; // if TRUE, the retain variables are initialized (warm start / cold start)
	bInCopyCode : BOOL;  // if TRUE, the instance afterwards gets moved into the copy code (online change)
	
	UnitID: STRING(80);
	UnitDescr: STRING(255); 
END_VAR
sID := UnitID;
sDescr := UnitDescr;
END_METHOD

METHOD setOff : BOOL
VAR_INPUT
END_VAR
eSMState := TURNING_OFF;
END_METHOD

METHOD setOn : BOOL
VAR_INPUT
END_VAR
eSMState := TURNING_ON;
END_METHOD

END_FUNCTION_BLOCK

// ---- POUs/01 Actuators/Dosing Machine/FB_Unit_RO_RND.TcPOU
{attribute 'OPC.UA.DA.StructuredType' := '1'}
FUNCTION_BLOCK FB_Unit_RO_RND EXTENDS FB_BaseDevice IMPLEMENTS I_Device

VAR
	bFirstRun: BOOL := TRUE;
	{attribute 'OPC.UA.DA' := '1'} 
	bOutContactor AT %Q*: BOOL := FALSE;
	
	
	{attribute 'OPC.UA.DA' := '0'} 
	eSMState: (WAIT, TURNING_ON, ON, TURNING_OFF, OFF);
	
	tDebounce: TIME := T#5S;
	fbTON_Debounce: TON := (PT := tDebounce, IN := FALSE);
	
END_VAR

fbTON_Debounce();

IF bFirstRun THEN
	fbTON_Debounce.IN := TRUE;
	bFirstRun := FALSE;
END_IF


IF GVL.bAutoUpdateDeviceState THEN
	eState := eStateTarget;	
END_IF


IF eMode = E_DeviceMode.MANUAL THEN
	bEnable := TRUE;
END_IF

IF bEnable AND eStateTarget = E_DeviceState.ON AND eState <> E_DeviceState.ON THEN
		eSMState := TURNING_ON;
END_IF

IF (bEnable = FALSE OR eStateTarget = E_DeviceState.OFF) AND eState <> E_DeviceState.OFF THEN
		eSMState := TURNING_OFF;
END_IF


CASE eSMState OF
	
	WAIT:
		//Wait for method call to change ESMState
		
	TURNING_ON: 
		IF fbTON_Debounce.Q THEN
			eState := E_DeviceState.TURNING_ON;
			bOutContactor := TRUE;
			fbTON_Debounce.IN := FALSE;
			eSMState := ON;
		END_IF

		
	ON:
		IF bOutContactor <> TRUE THEN
			raiseAlarm(Priority := E_AlarmPriority.High, Label := 'Power Lost', Enabled := TRUE, DeviceAlarmID := 1);
			eState := E_DeviceState.OFF;
			eSMState := TURNING_OFF;
		END_IF
			
	TURNING_OFF:
		fbTON_Debounce.IN := TRUE;
		bOutContactor := TRUE;
		eState := E_DeviceState.TURNING_OFF;
		bOutContactor := FALSE;
		eSMState := OFF;

	OFF:
		eState := E_DeviceState.OFF;
		eSMState := WAIT;
		fbTON_Debounce.IN := TRUE;
		
END_CASE

{warning 'add method implementation '}
METHOD disable : BOOL
bEnable := FALSE;
END_METHOD

{warning 'add method implementation '}
METHOD enable : BOOL
bEnable := TRUE;
END_METHOD

METHOD FB_init : BOOL
VAR_INPUT
	bInitRetains : BOOL; // if TRUE, the retain variables are initialized (warm start / cold start)
	bInCopyCode : BOOL;  // if TRUE, the instance afterwards gets moved into the copy code (online change)
	
	UnitID: STRING(80);
	UnitDescr: STRING(255); 
END_VAR
sID := UnitID;
sDescr := UnitDescr;
END_METHOD

METHOD setOff : BOOL
VAR_INPUT
END_VAR
eSMState := TURNING_OFF;
END_METHOD

METHOD setOn : BOOL
VAR_INPUT
END_VAR
eSMState := TURNING_ON;
END_METHOD

END_FUNCTION_BLOCK

// ---- POUs/01 Actuators/Dosing Machine/FB_UVFilter_Pentair_EU40.TcPOU
{attribute 'OPC.UA.DA.StructuredType' := '1'}
FUNCTION_BLOCK FB_UVFilter_Pentair_EU40 EXTENDS FB_BaseDevice IMPLEMENTS I_Device

VAR
	{attribute 'OPC.UA.DA' := '1'} 
	bInRelay AT %I*: BOOL := FALSE;
	
	{attribute 'OPC.UA.DA' := '1'} 
	bOutRelay AT %Q*: BOOL := FALSE;
	
	{attribute 'OPC.UA.DA' := '0'} 
	eSMState: (WAIT, TURNING_ON, ON, TURNING_OFF, OFF);
	
	{attribute 'OPC.UA.DA' := '0'} 
	tActionTimeout: TIME := T#5S;
	{attribute 'OPC.UA.DA' := '0'} 
	fbTON_timeout: TON := (PT := tActionTimeout, IN := FALSE);
END_VAR

IF GVL.bAutoUpdateDeviceState THEN
	eState := eStateTarget;	
END_IF

IF eMode = E_DeviceMode.MANUAL THEN
	bEnable := TRUE;
END_IF

IF (eStateTarget = E_DeviceState.ON) AND bEnable AND eSMState <> ON THEN
	eSMState := TURNING_ON;
END_IF

IF ((eStateTarget = E_DeviceState.OFF) OR (NOT bEnable)) AND eSMState <> OFF THEN
	eSMState := TURNING_OFF;
END_IF



CASE eSMState OF
	
		
	TURNING_ON: 
		bOutRelay := TRUE;
		eSMState := ON;
		eState := E_DeviceState.ON;
		
	ON:
		IF NOT bOutRelay THEN
			eSMState := TURNING_OFF;
		END_IF
		
	TURNING_OFF:
		bOutRelay := FALSE;
		eSMState := OFF;
		eState := E_DeviceState.TURNING_OFF;
		
	OFF:
		eState := E_DeviceState.OFF;
		bBusy := FALSE;
		
END_CASE

{warning 'add method implementation '}
METHOD disable : BOOL
bEnable := FALSE;
END_METHOD

{warning 'add method implementation '}
METHOD enable : BOOL
bEnable := TRUE;
END_METHOD

METHOD FB_init : BOOL
VAR_INPUT
	bInitRetains : BOOL; // if TRUE, the retain variables are initialized (warm start / cold start)
	bInCopyCode : BOOL;  // if TRUE, the instance afterwards gets moved into the copy code (online change)
	
	UnitID: STRING(80);
	UnitDescr: STRING(255); 
END_VAR
sID := UnitID;
sDescr := UnitDescr;
END_METHOD

METHOD setOff : BOOL
VAR_INPUT
END_VAR
IF bEnable THEN
	eSMState := TURNING_OFF;
END_IF
END_METHOD

METHOD setOn : BOOL
VAR_INPUT
END_VAR
IF bEnable THEN
	eSMState := TURNING_ON;
END_IF
END_METHOD

END_FUNCTION_BLOCK

// ---- POUs/01 Actuators/Dosing Machine/FB_UVFilter_UltraAqua_MR4_220PP.TcPOU
{attribute 'OPC.UA.DA.StructuredType' := '1'}
FUNCTION_BLOCK FB_UVFilter_UltraAqua_MR4_220PP EXTENDS FB_BaseDevice IMPLEMENTS I_Device

VAR
	{attribute 'OPC.UA.DA' := '1'} 
	bInContactor AT %I*: BOOL := FALSE;
	{attribute 'OPC.UA.DA' := '0'} 
	bInRun AT %I*: BOOL := FALSE;
	{attribute 'OPC.UA.DA' := '0'} 
	bInAlarm AT %I*: BOOL := FALSE;
	
	{attribute 'OPC.UA.DA' := '1'} 
	bOutContactor AT %Q*: BOOL := FALSE;
	{attribute 'OPC.UA.DA' := '0'} 
	bOutON AT %Q*: BOOL := FALSE;
	{attribute 'OPC.UA.DA' := '0'} 
	bOutEnable AT %Q*: BOOL := FALSE;
	
	{attribute 'OPC.UA.DA' := '0'} 
	eSMState: (WAIT, TURNING_ON, ON, TURNING_OFF, OFF);
	
	{attribute 'OPC.UA.DA' := '0'} 
	tActionTimeout: TIME := T#5S;
	{attribute 'OPC.UA.DA' := '0'} 
	fbTON_timeout: TON := (PT := tActionTimeout, IN := FALSE);
END_VAR

IF GVL.bAutoUpdateDeviceState THEN
	eState := eStateTarget;	
END_IF



CASE eSMState OF
	WAIT:
		//Wait for method call to change ESMState
	TURNING_ON: 
		bOutContactor := TRUE;
		bOutON := TRUE;
		bOutEnable := TRUE;
		eSMState := ON;
		eState := E_DeviceState.TURNING_ON;
	ON:
		IF bInContactor = TRUE AND bInRun = TRUE THEN
			eState := E_DeviceState.CLOSED;
			eSMState := ON;
			bBusy := FALSE;
		END_IF	
		
	TURNING_OFF:
		bOutContactor := FALSE;
		bOutEnable := FALSE;
		bOutON :=  FALSE;
		
		eSMState := OFF;
		eState := E_DeviceState.TURNING_OFF;
	OFF:
		IF bInContactor = FALSE AND bInRun = FALSE THEN
			eState := E_DeviceState.OFF;
			eSMState := WAIT;
			bBusy := FALSE;
		END_IF
END_CASE

{warning 'add method implementation '}
METHOD disable : BOOL
bEnable := FALSE;
END_METHOD

{warning 'add method implementation '}
METHOD enable : BOOL
bEnable := TRUE;
END_METHOD

METHOD FB_init : BOOL
VAR_INPUT
	bInitRetains : BOOL; // if TRUE, the retain variables are initialized (warm start / cold start)
	bInCopyCode : BOOL;  // if TRUE, the instance afterwards gets moved into the copy code (online change)
	
	UnitID: STRING(80);
	UnitDescr: STRING(255); 
END_VAR
sID := UnitID;
sDescr := UnitDescr;
END_METHOD

METHOD setOff : BOOL
VAR_INPUT
END_VAR
eSMState := TURNING_OFF;
END_METHOD

METHOD setOn : BOOL
VAR_INPUT
END_VAR
eSMState := TURNING_ON;
END_METHOD

END_FUNCTION_BLOCK

// ---- POUs/01 Actuators/FB_Valve_ONOFF_woMonitoring_1.TcPOU
{attribute 'OPC.UA.DA' := '1'}
FUNCTION_BLOCK FB_Valve_ONOFF_woMonitoring_1 EXTENDS FB_BaseDevice IMPLEMENTS I_Device, I_ValveActuated

VAR
	
	{attribute 'OPC.UA.DA' := '1'} 
	bValveMonitor_OPEN AT %I*: BOOL := FALSE;
	{attribute 'OPC.UA.DA' := '1'} 
	bValveMonitor_CLOSED AT %I*: BOOL := FALSE;
	{attribute 'OPC.UA.DA' := '1'} 
	bValveOutput_OPEN AT %Q*: BOOL := FALSE;
	{attribute 'OPC.UA.DA' := '1'} 
	bValveOutput_CLOSE AT %Q*: BOOL := FALSE;
	
	{attribute 'OPC.UA.DA' := '0'} 
	eSMState: (WAIT, CLOSING, CLOSED, OPENING, OPEN);
	
	{attribute 'OPC.UA.DA' := '1'} 
	tActionTimeout: TIME := T#5S;
	{attribute 'OPC.UA.DA' := '0'} 
	fbTON_timeout: TON := (PT := tActionTimeout, IN := FALSE);
	{attribute 'OPC.UA.DA' := '0'}
	fbTON_simulation_delay: TON := (PT := T#1S, IN := FALSE);
END_VAR

fbTONstartTime();
fbTONstopTime();

IF GVL.bAutoUpdateDeviceState THEN
	eState := eStateTarget;	
END_IF

IF bEnable = FALSE THEN
	eSMState := CLOSE
END_IF

	
CASE eSMState OF
	
	WAIT:
		//Wait for method call to change ESMState
		
	OPENING: 
		eState := E_DeviceState.TURNING_ON;
		bValveOutput_CLOSE 	:= FALSE;
		bValveOutput_OPEN 	:= TRUE;

	
		IF fbTONstartTime.Q THEN
			eSMState := WAIT;
			raiseAlarm(Priority := E_AlarmPriority.High, Label := 'Failed to Open', Enabled := TRUE, DeviceAlarmID := 1);
		END_IF
		
		IF bValveMonitor_OPEN  THEN
			eSMState := OPEN;
			eState := E_DeviceState.OPEN;
		END_IF
		
	OPEN:
		IF bValveMonitor_OPEN <> TRUE THEN
			raiseAlarm(Priority := E_AlarmPriority.High, Label := 'Valve Closed Unexpectedly', Enabled := TRUE, DeviceAlarmID := 2);
			eState := E_DeviceState.CLOSED;
			eSMState := WAIT;
		END_IF
		

	CLOSING:
		eState := E_DeviceState.TURNING_OFF;
		bValveOutput_CLOSE 	:= TRUE;
		bValveOutput_OPEN 	:= FALSE;

				
		IF fbTONstopTime.Q THEN
			eSMState := WAIT;
			raiseAlarm(Priority := E_AlarmPriority.High, Label := 'Failed to Close', Enabled := TRUE, DeviceAlarmID := 3);
		END_IF 
		
		IF bValveMonitor_CLOSED = TRUE THEN
			eSMState := CLOSED;	
		END_IF
		

	CLOSED:
		eState := E_DeviceState.CLOSED;
		eSMState := WAIT;
		
END_CASE

{warning 'add method implementation '}
METHOD close : BOOL
eSMState := CLOSING;
END_METHOD

{warning 'add method implementation '}
METHOD disable : BOOL
bEnable := FALSE;
END_METHOD

{warning 'add method implementation '}
METHOD enable : BOOL
bEnable := TRUE;
END_METHOD

{warning 'add method implementation '}
METHOD FB_init : BOOL
VAR_INPUT
	(* if TRUE, the retain variables are initialized (warm start / cold start)*)
	bInitRetains	: BOOL;
	(* if TRUE, the instance afterwards gets moved into the copy code (online change)*)
	bInCopyCode	: BOOL;
	
	ValveID: STRING(80);
	ValveDescr: STRING(255); 
END_VAR
sID := ValveID;
sDescr := ValveDescr;
END_METHOD

{warning 'add method implementation '}
METHOD open : BOOL
eSMState := OPENING;
END_METHOD

END_FUNCTION_BLOCK

// ---- POUs/01 Actuators/supersceded/FB_DosingPumpAgrowtek.TcPOU
{attribute 'OPC.UA.DA.StructuredType' := '1'}
FUNCTION_BLOCK FB_DosingPumpAgrowtek EXTENDS FB_BaseDevice IMPLEMENTS I_PumpDosing

VAR_IN_OUT
	{attribute 'OPC.UA.DA' := '0'}
	fbModbusMaster: FB_ModbusMaster;
END_VAR


VAR
	// Modbus Variables
	nPumpID: UINT;	
	nModbusUnitID: UINT; 
	ePumpType: E_DosingPump;
	
	{attribute 'OPC.UA.DA' := '0'}
	nReadRegsVals: ARRAY[1..10] OF WORD;
	{attribute 'OPC.UA.DA' := '0'}
	nWriteRegsVals: ARRAY[1..10] OF WORD;
	{attribute 'OPC.UA.DA' := '0'}
	nQtyWordsWrite: UINT;
	{attribute 'OPC.UA.DA' := '0'}
	nAddrWrite: UINT;
	{attribute 'OPC.UA.DA' := '0'}
	nRegisterWordstoRead: UINT;
	{attribute 'OPC.UA.DA' := '0'}
	nAddrRead: UINT;
	
	// Async Statemachine Variables
	{attribute 'OPC.UA.DA' := '0'}
	eSMState: (WAIT, READ_TRIG, READ, WRITE_TRIG, WRITE, SET_ON_TRIG, SET_ON, SET_OFF_TRIG, SET_OFF, ERROR);
	{attribute 'OPC.UA.DA' := '0'} 
	eOpType: (READ_OP, WRITE_OP);
	{attribute 'OPC.UA.DA' := '0'} 
	bRequestFinished: POINTER TO BOOL;
	{attribute 'OPC.UA.DA' := '0'} 
	bRequestSentToMaster: BOOL 	:= FALSE;
	{attribute 'OPC.UA.DA' := '0'} 
	bRequestCompleted: BOOL 	:= FALSE;
	
	// Dosing Variable
	{attribute 'OPC.UA.DA' := '0'} 
	fbTONdoseTime: TON;  // time the pump shall remain on at the nominated dosing rate
	{attribute 'OPC.UA.DA' := '0'} 
	fbTONdoseMsgDelay: TON := (PT := T#100MS); // ensures pump has sufficient time to respond to request
	{attribute 'OPC.UA.DA' := '1'} 
	nDoseRateMLph: UINT;
	{attribute 'OPC.UA.DA' := '1'} 
	nDoseQtyMls: UINT;
	{attribute 'OPC.UA.DA' := '1'} 
	tTimeToDose: TIME;
	{attribute 'OPC.UA.DA' := '1'} 
	nPumpSpeed: UINT; 
	
END_VAR

fbTONdoseTime();
fbTONdoseMsgDelay();

IF GVL.bAutoUpdateDeviceState THEN
	eState := eStateTarget;	
END_IF


CASE eSMState OF
	
	WAIT :
	//Do nothing and wait for eState to be changed by a called method

	READ_TRIG : //Read the first 122 registers (out of a total ~216)
	
		fbModbusMaster.readRegs(
			ReadRegsVals:= ADR(nReadRegsVals), 
			SlaveAddress:= nModbusUnitID, 
			QtyWordsToRead:= nRegisterWordstoRead, 
			AdrFirstSlaveRegisterRead:= nAddrRead, 
			bRequestCompleted:= ADR(bRequestCompleted), 
			bRequestAccepted=> bRequestSentToMaster);
				
		IF bRequestSentToMaster THEN
			eSMState := READ;				// set bBusy within the method calls
		END_IF
	
	READ:
		IF bRequestCompleted THEN	
			eSMState := WAIT; 			
			bRequestSentToMaster := FALSE;
			bRequestCompleted := FALSE;
			bBusy := FALSE;
		END_IF
		
		nPumpSpeed := nReadRegsVals[1];


	WRITE_TRIG :
		
		
		(* fbModbusMaster.writeRegs(
			WriteRegVals:= nWriteRegsVals, 
			SlaveAddress:= nModbusUnitID, 
			QtyWordsToWrite:= nQtyWordsWrite, 
			AdrFirstSlaveRegisterWrite:= nAddrWrite, 
			bRequestCompleted:= ADR(bRequestCompleted), 
			bRequestAccepted=> bRequestSentToMaster);
			*)
		
		fbModbusMaster.writeReg(
			WriteRegVal := nWriteRegsVals[1],
			SlaveAddress := nModbusUnitID,
			AdrFirstSlaveRegisterWrite := nAddrWrite,
			bRequestCompleted := ADR(bRequestCompleted),
			bRequestAccepted => bRequestSentToMaster);
			
			
		IF bRequestSentToMaster THEN
			eSMState := WRITE;           // set bBusy within the method calls
		END_IF
		
	
	WRITE:
		IF bRequestCompleted THEN
			eSMState := WAIT;
			bRequestCompleted := FALSE;
			bRequestSentToMaster := FALSE;
			bBusy := FALSE;
		END_IF
		
		
	
	SET_ON_TRIG:
		(*
		fbModbusMaster.writeRegs(
			WriteRegVals:= nWriteRegsVals, 
			SlaveAddress:= nModbusUnitID, 
			QtyWordsToWrite:= 1, 				
			AdrFirstSlaveRegisterWrite:= nAddrWrite, 
			bRequestCompleted:= ADR(bRequestCompleted), 
			bRequestAccepted=> bRequestSentToMaster);
			*)
			
		fbModbusMaster.writeReg(
			WriteRegVal := nWriteRegsVals[1],
			SlaveAddress := nModbusUnitID,
			AdrFirstSlaveRegisterWrite := nAddrWrite,
			bRequestCompleted := ADR(bRequestCompleted),
			bRequestAccepted => bRequestSentToMaster);
			
		eSMState := SET_ON;
		
	SET_ON:
		IF bRequestCompleted  THEN
			eSMState := SET_OFF_TRIG;
			bRequestCompleted := FALSE;
			bRequestSentToMaster := FALSE;
			fbTONdoseTime(IN:=TRUE, PT := tTimeToDose); // start the min delay timer and dose timer
			fbTONdoseMsgDelay(IN:= TRUE);			 
		END_IF	
	
	
		
		
	SET_OFF_TRIG:
	      
		IF fbModbusMaster.isBusy() = FALSE THEN
			IF fbTONdoseMsgDelay.Q AND fbTONdoseTime.Q THEN
		
				fbModbusMaster.writeReg(
					WriteRegVal := 0, // turn off
					SlaveAddress := nModbusUnitID,
					AdrFirstSlaveRegisterWrite := nAddrWrite,
					bRequestCompleted := ADR(bRequestCompleted),
					bRequestAccepted => bRequestSentToMaster);
				
				(*
				nWriteRegsVals[1] := 0; // set the speed to 0
				fbModbusMaster.writeRegs(
					WriteRegVals:= nWriteRegsVals, 
					SlaveAddress:= nModbusUnitID, 
					QtyWordsToWrite:= 1, 				
					AdrFirstSlaveRegisterWrite:= nAddrWrite, 
					bRequestCompleted:= ADR(bRequestCompleted), 
					bRequestAccepted=> bRequestSentToMaster);
					*)
				fbTONdoseMsgDelay.IN := FALSE;
				fbTONdoseTime.IN := FALSE;
				eSMState := SET_OFF;
			END_IF
		END_IF
		
		
		
	SET_OFF:
		IF bRequestCompleted THEN
			eSMState := WAIT;
			bRequestCompleted := FALSE;
			bRequestSentToMaster := FALSE;
			bBusy := FALSE;
			nDoseQtyMls := 0;  // Set this to zero so that the historised tag can capture duplicate successive doses
		END_IF
		
END_CASE

{warning 'add method implementation '}
METHOD executeDose : BOOL
VAR_INPUT
	DoseQtyMls	: LREAL;
	DoseRateMlph: UINT; // ignore this (required to comply to interface)
	RequestComplete	: POINTER TO BOOL;
END_VAR
VAR_OUTPUT
	RequestAccepted	: BOOL;
END_VAR
(* setDose dispenses the amount requested at a user requested dose rate *)
(*
IF NOT bBusy AND bEnable THEN
		nDoseQtyMls := DoseQtyMls;
		nDoseRateMLph := DoseQtyMls;
		tTimeToDose := REAL_TO_TIME( (((UINT_TO_REAL(nDoseQtyMls)) / 480) * 60.0)*1000);  // Agrowtek maximum flow rate is 480 ml/min
		nWriteRegsVals[1] := 100;
		nAddrWrite := getAdrReadWriteSpeed(ePumpType);
		bBusy := TRUE;
		RequestAccepted := TRUE;
		bRequestSentToMaster := FALSE;
		bRequestFinished := RequestComplete;
		eSMState := SET_ON_TRIG;
		bBusy := TRUE;
END_IF
*)
END_METHOD

METHOD FB_init : BOOL


VAR_INPUT
	bInitRetains : BOOL; // if TRUE, the retain variables are initialized (warm start / cold start)
	bInCopyCode : BOOL;  // if TRUE, the instance afterwards gets moved into the copy code (online change)
	
	PumpID: STRING;
	PumpDescription: STRING;
	PumpType: E_DosingPump;
	
	
END_VAR
sID := PumpID;
sDescr := PumpDescription;
ePumpType := PumpType;
END_METHOD

METHOD getAdrReadAccumRunTime : BOOL
VAR_INPUT
	PumpType: E_DosingPump;
END_VAR
// This method retrieves the Modbus register for the individual Agrowtek pump
// We need to do this because 5 pumps share the same Modbus slave ID, however have differing registers to write to

CASE PumpType OF
	
	E_DosingPump.PH_UP:
		nAddrWrite := 16#64;
		
	E_DosingPump.PH_DOWN:
		nAddrWrite := 16#65;
		
	E_DosingPump.NUTRIENT_A:
		nAddrWrite := 16#66;
		
	E_DosingPump.NUTRIENT_B:
		nAddrWrite := 16#67;
		
	E_DosingPump.NUTRIENT_C:
		nAddrWrite := 16#68;
		
END_CASE
END_METHOD

METHOD getAdrReadWriteSpeed : UINT
VAR_INPUT
	PumpType: E_DosingPump;
END_VAR
// This method retrieves the Modbus register for the individual Agrowtek pump
// We need to do this because 5 pumps share the same Modbus slave ID, however have differing registers to write to

CASE PumpType OF
	
	E_DosingPump.PH_UP:
		getAdrReadWriteSpeed := 16#64;
		
	E_DosingPump.PH_DOWN:
		getAdrReadWriteSpeed := 16#65;
		
	E_DosingPump.NUTRIENT_A:
		getAdrReadWriteSpeed := 16#66;
		
	E_DosingPump.NUTRIENT_B:
		getAdrReadWriteSpeed := 16#67;
		
	E_DosingPump.NUTRIENT_C:
		getAdrReadWriteSpeed := 16#68;
		
END_CASE
END_METHOD

METHOD readSpeed : BOOL
VAR_INPUT
	RequestComplete	: POINTER TO BOOL;
	AddressToRead: UINT;
	NumberWords: UINT;
END_VAR
VAR_OUTPUT
	RequestAccepted	: BOOL;
END_VAR
IF NOT bBusy AND bEnable THEN
	nReadRegsVals[1] := 16#00;
	nReadRegsVals[2] := 16#00;
	nReadRegsVals[3] := 16#00;
	nReadRegsVals[4] := 16#00;
	nRegisterWordstoRead := NumberWords;
	nAddrRead:= AddressToRead;
	eSMState := READ_TRIG;
	bBusy := TRUE;		
	readSpeed := TRUE;		
ELSE
	readSpeed := FALSE;
END_IF
END_METHOD

METHOD setModID : BOOL
VAR_INPUT
	desiredID: UINT;
END_VAR
IF NOT bBusy AND bEnable THEN
	nModbusUnitID := 254;
	nQtyWordsWrite := 1;
	nAddrWrite := 0;
	nWriteRegsVals[1] := desiredID; 
	eSMState := WRITE_TRIG;
END_IF
END_METHOD

{warning 'add method implementation '}
METHOD setOFF : BOOL
VAR_INPUT
	RequestComplete	: POINTER TO BOOL;
END_VAR
VAR_OUTPUT
	RequestAccepted	: BOOL;
END_VAR
IF NOT bBusy AND bEnable THEN
	nModbusUnitID := 3;
	nWriteRegsVals[1] := 16#0; // speed 0
	nQtyWordsWrite := 1;
	nAddrWrite := getAdrReadWriteSpeed(ePumpType);
	eSMState := WRITE_TRIG;
	RequestAccepted := TRUE;
	bRequestSentToMaster := FALSE;
	bRequestFinished := RequestComplete;
	bBusy := TRUE;
	setOFF := TRUE;
ELSE
	setOFF := FALSE;
END_IF
END_METHOD

METHOD setOFF_All : BOOL
VAR_INPUT
	RequestComplete	: POINTER TO BOOL;
END_VAR
VAR_OUTPUT
	RequestAccepted	: BOOL;
END_VAR
IF NOT bBusy AND bEnable THEN
	nModbusUnitID := 3;
	nWriteRegsVals[1] := 100; // speed 100
	nWriteRegsVals[2] := 100; // speed 100
	nWriteRegsVals[3] := 100; // speed 100
	nWriteRegsVals[4] := 100; // speed 100
	nWriteRegsVals[5] := 100; // speed 100
	nQtyWordsWrite := 5;
	nAddrWrite := 100;
	eSMState := WRITE_TRIG;
	RequestAccepted := TRUE;
	bRequestSentToMaster := FALSE;
	bRequestFinished := RequestComplete;

	setOFF_All := TRUE;
ELSE
	setOFF_All := FALSE;
END_IF
END_METHOD

{warning 'add method implementation '}
METHOD setON : BOOL
VAR_INPUT
	RateMlph	: UINT;
	RequestComplete	: POINTER TO BOOL;
END_VAR
VAR_OUTPUT
	RequestAccepted	: BOOL;
END_VAR
IF NOT bBusy AND bEnable THEN
	nModbusUnitID := 3;
	nWriteRegsVals[1] := 16#64; // speed 100
	nQtyWordsWrite := 2;
	nAddrWrite := getAdrReadWriteSpeed(ePumpType);
	eSMState := WRITE_TRIG;
	RequestAccepted := TRUE;
	bRequestSentToMaster := FALSE;
	bRequestFinished := RequestComplete;
	bBusy := TRUE;
	setON := TRUE;
ELSE
	setON := FALSE;
END_IF
END_METHOD

METHOD setON_All : BOOL
VAR_INPUT
	RequestComplete	: POINTER TO BOOL;
END_VAR
VAR_OUTPUT
	RequestAccepted	: BOOL;
END_VAR
IF NOT bBusy AND bEnable THEN
	nModbusUnitID := 3;
	nWriteRegsVals[1] := 0; // speed 0
	nWriteRegsVals[2] := 0; // speed 0
	nWriteRegsVals[3] := 0; // speed 0
	nWriteRegsVals[4] := 0; // speed 0
	nWriteRegsVals[5] := 0; // speed 0
	nQtyWordsWrite := 5;
	nAddrWrite := 100;
	eSMState := WRITE_TRIG;
	RequestAccepted := TRUE;
	bRequestSentToMaster := FALSE;
	bRequestFinished := RequestComplete;

	setON_All := TRUE;
ELSE
	setON_All := FALSE;
END_IF
END_METHOD

END_FUNCTION_BLOCK

// ---- POUs/02 Sensors/Dosing Machine/FB_Sensor_AtlasDO.TcPOU
{attribute 'OPC.UA.DA' := '1'}
FUNCTION_BLOCK FB_Sensor_AtlasDO EXTENDS FB_BaseDevice IMPLEMENTS I_Device, I_Sensor

VAR
	
	{attribute 'OPC.UA.DA' := '0'} 
	eSensorType: E_SensorType;
	{attribute 'OPC.UA.DA' := '0'}
	nRawInput AT %I*: INT;
	nFaultInput AT %I*: BOOL;
	{attribute 'OPC.UA.DA' := '1'}
	nCurrentValue: REAL;
	
	{attribute 'OPC.UA.DA' := '0'} 
	nCalOutputLOW AT %Q*: BOOL;
	{attribute 'OPC.UA.DA' := '0'} 
	nCalOutputHIGH AT %Q*: BOOL;
	
	{attribute 'OPC.UA.DA' := '0'} 
	trigCalibrate: R_TRIG;
	
	{attribute 'OPC.UA.DA' := '0'} 
	timerBtnPress: TON := (PT:=T#250MS,IN := FALSE);
	{attribute 'OPC.UA.DA' := '0'} 
	timerDoCalibration: TON := (PT:=T#120S,IN := FALSE); // Check this time during testing! The instructions are not clear about what happens after initiating a calibration request 
	{attribute 'OPC.UA.DA' := '0'} 
	eSMState: (WAIT, LOW_START, LOW_END, HIGH_START, HIGH_END) := WAIT;
	
END_VAR

calculate();
trigCalibrate();
timerBtnPress();


CASE eSMState OF 
	WAIT:
		// wait for the calibrate method call to change the ESMState variable
		

	LOW_START:
		nCalOutputLOW := TRUE;
		timerBtnPress.IN := TRUE;
		IF timerBtnPress.Q THEN
			nCalOutputLOW := FALSE;
			eSMState := LOW_END;
			timerBtnPress.IN := FALSE; 
			timerDoCalibration.IN := TRUE;
		END_IF
		
		eSMState := LOW_END;
		
	LOW_END:
		IF timerDoCalibration.Q THEN
			timerDoCalibration.IN := FALSE;
			bBusy := FALSE;
			eSMState := WAIT;
		END_IF
	
	
	HIGH_START:
		nCalOutputHIGH := TRUE;
		timerBtnPress.IN := TRUE;
		IF timerBtnPress.Q THEN
			nCalOutputHIGH := FALSE;
			eSMState := HIGH_END;
			timerBtnPress.IN := FALSE; 
			timerDoCalibration.IN := TRUE;
		END_IF
		
		eSMState := HIGH_END;
		
	HIGH_END:
		IF timerDoCalibration.Q THEN
			timerDoCalibration.IN := FALSE;
			bBusy := FALSE;
			eSMState := WAIT;
		END_IF
		

END_CASE

METHOD PRIVATE calculate : BOOL
VAR_INPUT
	
	// Var
END_VAR
VAR
	nMeasuredCurrent: REAL;
END_VAR
nMeasuredCurrent := (INT_TO_REAL(nRawInput)/GVL.nMaxADCOutput)*16.0 + 4.0; // in mA


// nCurrentValue := (nMeasuredCurrent - 4.0) * 2.0;  // equation is DO = (mA reading - 4.0) / 0.5

nCurrentValue := (nMeasuredCurrent - 4.0) * 2.0;  // equation is DO = (mA reading - 4.0) / 0.5
END_METHOD

METHOD calibrate : BOOL
VAR_INPUT
	TestType: INT; // LOW = 1, HIGH = 2
END_VAR
CASE TestType OF
	1:
		eSMState := LOW_START;
	2:
		eSMState := HIGH_START;
		
END_CASE

bBusy := TRUE;
END_METHOD

{warning 'add method implementation '}
METHOD disable : BOOL
bEnable := FALSE;
END_METHOD

{warning 'add method implementation '}
METHOD enable : BOOL
bEnable := TRUE;
END_METHOD

{warning 'add method implementation '}
METHOD FB_init : BOOL
VAR_INPUT
	(* if TRUE, the retain variables are initialized (warm start / cold start)*)
	bInitRetains	: BOOL;
	(* if TRUE, the instance afterwards gets moved into the copy code (online change)*)
	bInCopyCode	: BOOL;
	
	SensorID	: STRING(80);
	SensorDescr	: STRING(255);
	SensorType	: E_SensorType;
END_VAR
sID := SensorID;
sDescr := SensorDescr;
eSensorType := SensorType;
END_METHOD

{warning 'add method implementation '}
METHOD getType : E_SensorType
getType := eSensorType;
END_METHOD

{warning 'add method implementation '}
METHOD getValue : REAL
getValue := nCurrentValue;
END_METHOD

{warning 'add method implementation '}
METHOD write : BOOL
// use this method to initiated a hardware read from assigned IO if required
END_METHOD

END_FUNCTION_BLOCK

// ---- POUs/02 Sensors/Dosing Machine/FB_Sensor_AtlasEC.TcPOU
{attribute 'OPC.UA.DA.StructuredType' := '1'}
FUNCTION_BLOCK FB_Sensor_AtlasEC EXTENDS FB_BaseDevice IMPLEMENTS I_Device, I_Sensor

VAR

	{attribute 'OPC.UA.DA' := '0'} 
	eSensorType: E_SensorType;
	nRawInput AT %I*: INT;
	nFaultInput AT %I*: BOOL;
	nCurrentValue: REAL;
	
	{attribute 'OPC.UA.DA' := '0'} 
	nCalOutputDRY AT %Q*: BOOL;
	{attribute 'OPC.UA.DA' := '0'} 
	nCalOutputLOW AT %Q*: BOOL;
	{attribute 'OPC.UA.DA' := '0'} 
	nCalOutputHIGH AT %Q*: BOOL;
	{attribute 'OPC.UA.DA' := '0'} 	
	trigCalibrate: R_TRIG;
	{attribute 'OPC.UA.DA' := '0'} 
	timerBtnPress: TON := (PT:=T#250MS,IN := FALSE);
	{attribute 'OPC.UA.DA' := '0'} 
	timerDoCalibration: TON := (PT:=T#120S,IN := FALSE); // Check this time during testing! The instructions are not clear about what happens after initiating a calibration request 
	{attribute 'OPC.UA.DA' := '0'} 
	eSMState: (WAIT, DRY_START, DRY_END, LOW_START, LOW_END, HIGH_START, HIGH_END) := WAIT;
	
	
	
END_VAR

calculate();
trigCalibrate();
timerBtnPress();

CASE eSMState OF 
	WAIT:
		// wait for the calibrate method call to change the ESMState variable
		
	DRY_START:
		nCalOutputDRY := TRUE;
		timerBtnPress.IN := TRUE;
		IF timerBtnPress.Q THEN
			nCalOutputDRY := FALSE;
			eSMState := DRY_END;
			timerBtnPress.IN := FALSE; 
			timerDoCalibration.IN := TRUE;
		END_IF
		
		eSMState := DRY_END;
		
	DRY_END:
		IF timerDoCalibration.Q THEN
			timerDoCalibration.IN := FALSE;			// CHeck the functionality of this step - instructions are not clear
			bBusy := FALSE;
			eSMState := WAIT;
		END_IF
		
	LOW_START:
		nCalOutputLOW := TRUE;
		timerBtnPress.IN := TRUE;
		IF timerBtnPress.Q THEN
			nCalOutputLOW := FALSE;
			eSMState := LOW_END;
			timerBtnPress.IN := FALSE; 
			timerDoCalibration.IN := TRUE;
		END_IF
		
		eSMState := LOW_END;
		
	LOW_END:
		IF timerDoCalibration.Q THEN
			timerDoCalibration.IN := FALSE;
			bBusy := FALSE;
			eSMState := WAIT;
		END_IF
	
	
	HIGH_START:
		nCalOutputHIGH := TRUE;
		timerBtnPress.IN := TRUE;
		IF timerBtnPress.Q THEN
			nCalOutputHIGH := FALSE;
			eSMState := HIGH_END;
			timerBtnPress.IN := FALSE; 
			timerDoCalibration.IN := TRUE;
		END_IF
		
		eSMState := HIGH_END;
		
	HIGH_END:
		IF timerDoCalibration.Q THEN
			timerDoCalibration.IN := FALSE;
			bBusy := FALSE;
			eSMState := WAIT;
		END_IF

END_CASE

METHOD PRIVATE calculate : BOOL
VAR_INPUT
	
	// Var
END_VAR

VAR
	nMeasuredCurrent: REAL;
END_VAR
nMeasuredCurrent := (INT_TO_REAL(nRawInput)/GVL.nMaxADCOutput)*16.0 + 4.0; // in mA

//nCurrentValue := (nMeasuredCurrent - 4.0) / 0.004; // this equation for a K0.1 probe - there are other types of probes available

// nCurrentValue := (nMeasuredCurrent - 4.0) / 0.004; // this equation for a K0.1 probe - there are other types of probes available


nCurrentValue := ((nMeasuredCurrent - 4.0) / 0.004) / 1000.0; // this equation for a K0.1 probe - there are other types of probes available
END_METHOD

METHOD calibrate : BOOL
VAR_INPUT
	TestType: INT; // DRY = 1, LOW = 2, HIGH = 3
END_VAR
CASE TestType OF
	1:
		eSMState := DRY_START;
	2:
		eSMState := LOW_START;
	3:
		eSMState := HIGH_START;
END_CASE

bBusy := TRUE;
END_METHOD

{warning 'add method implementation '}
METHOD disable : BOOL
bEnable := FALSE;
END_METHOD

{warning 'add method implementation '}
METHOD enable : BOOL
bEnable := TRUE;
END_METHOD

{warning 'add method implementation '}
METHOD FB_init : BOOL
VAR_INPUT
	(* if TRUE, the retain variables are initialized (warm start / cold start)*)
	bInitRetains	: BOOL;
	(* if TRUE, the instance afterwards gets moved into the copy code (online change)*)
	bInCopyCode	: BOOL;
	
	SensorID	: STRING(80);
	SensorDescr	: STRING(255);
	SensorType	: E_SensorType;
END_VAR
sID := SensorID;
sDescr := SensorDescr;
eSensorType := SensorType;
END_METHOD

{warning 'add method implementation '}
METHOD getType : E_SensorType
getType := eSensorType;
END_METHOD

{warning 'add method implementation '}
METHOD getValue : REAL
getValue := nCurrentValue;
END_METHOD

{warning 'add method implementation '}
METHOD write : BOOL
// use this method to initiated a hardware read from assigned IO if required
END_METHOD

END_FUNCTION_BLOCK

// ---- POUs/02 Sensors/Dosing Machine/FB_Sensor_AtlasORP.TcPOU
{attribute 'OPC.UA.DA.StructuredType' := '1'}
FUNCTION_BLOCK FB_Sensor_AtlasORP EXTENDS FB_BaseDevice IMPLEMENTS I_Device, I_Sensor

VAR
	{attribute 'OPC.UA.DA' := '0'} 	
	eSensorType: E_SensorType;
	{attribute 'OPC.UA.DA' := '0'}
	nRawInput AT %I*: INT;
	nFaultInput AT %I*: BOOL;
	{attribute 'OPC.UA.DA' := '1'}
	nCurrentValue: REAL;
	{attribute 'OPC.UA.DA' := '0'} 
	nCalOutputCAL AT %Q*: BOOL;

	{attribute 'OPC.UA.DA' := '0'} 
	trigCalibrate: R_TRIG;
	{attribute 'OPC.UA.DA' := '0'} 
	timerBtnPress: TON := (PT:=T#250MS,IN := FALSE);
	{attribute 'OPC.UA.DA' := '0'} 
	timerDoCalibration: TON := (PT:=T#120S,IN := FALSE); // Check this time during testing! The instructions are not clear about what happens after initiating a calibration request 
	{attribute 'OPC.UA.DA' := '0'} 
	eSMState: (WAIT, CAL_START, CAL_END) := WAIT;
	
	
END_VAR

calculate();
trigCalibrate();
timerBtnPress();

CASE eSMState OF 
	WAIT:
		// wait for the calibrate method call to change the ESMState variable
		
	CAL_START:
		nCalOutputCAL := TRUE;
		timerBtnPress.IN := TRUE;
		IF timerBtnPress.Q THEN
			nCalOutputCAL := FALSE;
			eSMState := CAL_END;
			timerBtnPress.IN := FALSE; 
			timerDoCalibration.IN := TRUE;
		END_IF
		
		eSMState := CAL_END;
		
	CAL_END:
		IF timerDoCalibration.Q THEN
			timerDoCalibration.IN := FALSE;			// CHeck the functionality of this step - instructions are not clear
			bBusy := FALSE;
			eSMState := WAIT;
		END_IF
		
END_CASE

METHOD PRIVATE calculate : BOOL
VAR_INPUT
	
	// Var
END_VAR
VAR
	nMeasuredCurrent: REAL;
END_VAR
nMeasuredCurrent := (INT_TO_REAL(nRawInput)/GVL.nMaxADCOutput)*16.0 + 4.0; // in mA

nCurrentValue := ((nMeasuredCurrent - 12.0) / 8.0) * 1900.0;
END_METHOD

METHOD calibrate : BOOL
VAR_INPUT
			// No input needed as it is a 1 stage calibration
END_VAR
eSMState := CAL_START;
bBusy := TRUE;
END_METHOD

{warning 'add method implementation '}
METHOD disable : BOOL
bEnable := FALSE;
END_METHOD

{warning 'add method implementation '}
METHOD enable : BOOL
bEnable := TRUE;
END_METHOD

{warning 'add method implementation '}
METHOD FB_init : BOOL
VAR_INPUT
	(* if TRUE, the retain variables are initialized (warm start / cold start)*)
	bInitRetains	: BOOL;
	(* if TRUE, the instance afterwards gets moved into the copy code (online change)*)
	bInCopyCode	: BOOL;
	
	SensorID	: STRING(80);
	SensorDescr	: STRING(255);
	SensorType	: E_SensorType;
END_VAR
sID := SensorID;
sDescr := SensorDescr;
eSensorType := SensorType;
END_METHOD

{warning 'add method implementation '}
METHOD getType : E_SensorType
getType := eSensorType;
END_METHOD

{warning 'add method implementation '}
METHOD getValue : REAL
getValue := nCurrentValue;
END_METHOD

{warning 'add method implementation '}
METHOD write : BOOL
// use this method to initiated a hardware read from assigned IO if required
END_METHOD

END_FUNCTION_BLOCK

// ---- POUs/02 Sensors/Dosing Machine/FB_Sensor_AtlasPH.TcPOU
{attribute 'OPC.UA.DA.StructuredType' := '1'}
FUNCTION_BLOCK FB_Sensor_AtlasPH EXTENDS FB_BaseDevice IMPLEMENTS I_Device, I_Sensor

VAR

	{attribute 'OPC.UA.DA' := '0'} 
	eSensorType: E_SensorType;
	{attribute 'OPC.UA.DA' := '0'} 
	nRawInput AT %I*: INT;
	nFaultInput AT %I*: BOOL;
	{attribute 'OPC.UA.DA' := '1'} 
	nCurrentValue: REAL;
	
	{attribute 'OPC.UA.DA' := '0'} 
	nCalOutputPH7 AT %Q*: BOOL;
	{attribute 'OPC.UA.DA' := '0'} 
	nCalOutputPH4 AT %Q*: BOOL;
	{attribute 'OPC.UA.DA' := '0'} 
	nCalOutputPH10 AT %Q*: BOOL;
	
	{attribute 'OPC.UA.DA' := '0'} 
	trigCalibrate: R_TRIG;
	{attribute 'OPC.UA.DA' := '0'} 
	timerBtnPress: TON := (PT:=T#250MS,IN := FALSE);
	
	{attribute 'OPC.UA.DA' := '0'} 
	timerDoCalibration: TON := (PT:=T#120S,IN := FALSE); // Check this time during testing! The instructions are not clear about what happens after initiating a calibration request 
	
	{attribute 'OPC.UA.DA' := '0'} 
	eSMState: (WAIT, pH_7_START, pH_7_END, pH_4_START, pH_4_END, pH_10_START, pH_10_END) := WAIT;
END_VAR

calculate();
trigCalibrate();
timerBtnPress();

CASE eSMState OF 
	WAIT:
		// wait for the calibrate method call to change the ESMState variable
		
	pH_7_START:
		nCalOutputPH7 := TRUE;
		timerBtnPress.IN := TRUE;
		IF timerBtnPress.Q THEN
			nCalOutputPH7 := FALSE;
			eSMState := pH_7_END;
			timerBtnPress.IN := FALSE; 
			timerDoCalibration.IN := TRUE;
		END_IF
		
		eSMState := pH_7_END;
		
	pH_7_END:
		IF timerDoCalibration.Q THEN
			timerDoCalibration.IN := FALSE;			// CHeck the functionality of this step - instructions are not clear
			bBusy := FALSE;
			eSMState := WAIT;
		END_IF
		
	pH_4_START:
		nCalOutputPH4 := TRUE;
		timerBtnPress.IN := TRUE;
		IF timerBtnPress.Q THEN
			nCalOutputPH4 := FALSE;
			eSMState := pH_4_END;
			timerBtnPress.IN := FALSE; 
			timerDoCalibration.IN := TRUE;
		END_IF
		
		eSMState := pH_4_END;
		
